// ---- DUTs/IO/PdoEntries/FSOE_340991D3.TcDUT
{attribute addProperty BoxType "EK1960-2600-0019"}
{attribute addProperty Id "FSoE_CommandUSINT811FSOUT_Module_1_Channel_1_OutputBIT10.1251FSOUT_Module_1_Channel_2_OutputBIT10.1252FSOUT_Module_1_Channel_3_OutputBIT10.1253FSOUT_Module_1_Channel_4_OutputBIT10.1254FSOUT_Module_1_ErrAckBIT10.1251FSOUT_Module_2_Channel_1_OutputBIT10.1251FSOUT_Module_2_Channel_2_OutputBIT10.1252FSOUT_Module_2_Channel_3_OutputBIT10.1253FSOUT_Module_2_Channel_4_OutputBIT10.1254FSOUT_Module_2_ErrAckBIT10.1251FSOUT_Module_3_Channel_1_OutputBIT10.1251FSOUT_Module_3_Channel_2_OutputBIT10.1252FSOUT_Module_3_Channel_3_OutputBIT10.1253FSOUT_Module_3_Channel_4_OutputBIT10.1254FSOUT_Module_3_ErrAckBIT10.1251FSOUT_Module_4_Channel_1_OutputBIT10.1251FSoE_CRC_000UINT1623FSOUT_Module_4_Channel_2_OutputBIT10.1252FSOUT_Module_4_Channel_3_OutputBIT10.1253FSOUT_Module_4_Channel_4_OutputBIT10.1254FSOUT_Module_4_ErrAckBIT10.1251FSOUT_Module_5_Channel_1_OutputBIT10.1251FSOUT_Module_5_Channel_2_OutputBIT10.1252FSOUT_Module_5_Channel_3_OutputBIT10.1253FSOUT_Module_5_Channel_4_OutputBIT10.1254FSOUT_Module_5_ErrAckBIT10.1251FSOUT_Module_6_Channel_1_OutputBIT10.1251FSOUT_Module_6_Channel_2_OutputBIT10.1252FSOUT_Module_6_Channel_3_OutputBIT10.1253FSOUT_Module_6_Channel_4_OutputBIT10.1254FSOUT_Module_6_ErrAckBIT10.1251FSOUT_Relais_Module_Channel_1_OutputBIT10.1251FSOUT_Relais_Module_Channel_2_OutputBIT10.1252FSoE_CRC_001UINT1624FSOUT_Relais_Module_Channel_3_OutputBIT10.1253FSOUT_Relais_Module_Channel_4_OutputBIT10.1254FSOUT_Relais_Module_ErrAckBIT10.1251FSIN_Module_1_ErrAckBIT10.1251FSIN_Module_2_ErrAckBIT10.1251FSIN_Module_3_ErrAckBIT10.1251FSIN_Module_4_ErrAckBIT10.1251FSIN_Module_5_ErrAckBIT10.1251FSIN_Module_6_ErrAckBIT10.1251FSIN_Module_7_ErrAckBIT10.1251FSIN_Module_8_ErrAckBIT10.1251FSIN_Module_9_ErrAck_1BIT10.1251FSIN_Module_9_ErrAck_2BIT10.1252FSIN_Module_10_ErrAck_1BIT10.1251FSIN_Module_10_ErrAck_2BIT10.1252FSoE_CRC_002UINT1625FSoE_Connection_IDUINT1622"}
{attribute addProperty CRC "873042387"}
{attribute addProperty SizeInBites "120"}
{attribute addProperty SizeInBytes "15"}
TYPE FSOE_340991D3 :
STRUCT
	{attribute addProperty Name "FSoE_Command"}
	FSoE_Command : USINT;
	{attribute addProperty Name "FSOUT_Module_1_Channel_1_Output"}
	FSOUT_Module_1_Channel_1_Output : BOOL;
	{attribute addProperty Name "FSOUT_Module_1_Channel_2_Output"}
	FSOUT_Module_1_Channel_2_Output : BOOL;
	{attribute addProperty Name "FSOUT_Module_1_Channel_3_Output"}
	FSOUT_Module_1_Channel_3_Output : BOOL;
	{attribute addProperty Name "FSOUT_Module_1_Channel_4_Output"}
	FSOUT_Module_1_Channel_4_Output : BOOL;
	{attribute addProperty Name "FSOUT_Module_1_ErrAck"}
	FSOUT_Module_1_ErrAck : BOOL;
	{attribute addProperty Name "FSOUT_Module_2_Channel_1_Output"}
	FSOUT_Module_2_Channel_1_Output : BOOL;
	{attribute addProperty Name "FSOUT_Module_2_Channel_2_Output"}
	FSOUT_Module_2_Channel_2_Output : BOOL;
	{attribute addProperty Name "FSOUT_Module_2_Channel_3_Output"}
	FSOUT_Module_2_Channel_3_Output : BOOL;
	{attribute addProperty Name "FSOUT_Module_2_Channel_4_Output"}
	FSOUT_Module_2_Channel_4_Output : BOOL;
	{attribute addProperty Name "FSOUT_Module_2_ErrAck"}
	FSOUT_Module_2_ErrAck : BOOL;
	{attribute addProperty Name "FSOUT_Module_3_Channel_1_Output"}
	FSOUT_Module_3_Channel_1_Output : BOOL;
	{attribute addProperty Name "FSOUT_Module_3_Channel_2_Output"}
	FSOUT_Module_3_Channel_2_Output : BOOL;
	{attribute addProperty Name "FSOUT_Module_3_Channel_3_Output"}
	FSOUT_Module_3_Channel_3_Output : BOOL;
	{attribute addProperty Name "FSOUT_Module_3_Channel_4_Output"}
	FSOUT_Module_3_Channel_4_Output : BOOL;
	{attribute addProperty Name "FSOUT_Module_3_ErrAck"}
	FSOUT_Module_3_ErrAck : BOOL;
	{attribute addProperty Name "FSOUT_Module_4_Channel_1_Output"}
	FSOUT_Module_4_Channel_1_Output : BOOL;
	{attribute addProperty Name "FSoE_CRC_000"}
	FSoE_CRC_000 : UINT;
	{attribute addProperty Name "FSOUT_Module_4_Channel_2_Output"}
	FSOUT_Module_4_Channel_2_Output : BOOL;
	{attribute addProperty Name "FSOUT_Module_4_Channel_3_Output"}
	FSOUT_Module_4_Channel_3_Output : BOOL;
	{attribute addProperty Name "FSOUT_Module_4_Channel_4_Output"}
	FSOUT_Module_4_Channel_4_Output : BOOL;
	{attribute addProperty Name "FSOUT_Module_4_ErrAck"}
	FSOUT_Module_4_ErrAck : BOOL;
	{attribute addProperty Name "FSOUT_Module_5_Channel_1_Output"}
	FSOUT_Module_5_Channel_1_Output : BOOL;
	{attribute addProperty Name "FSOUT_Module_5_Channel_2_Output"}
	FSOUT_Module_5_Channel_2_Output : BOOL;
	{attribute addProperty Name "FSOUT_Module_5_Channel_3_Output"}
	FSOUT_Module_5_Channel_3_Output : BOOL;
	{attribute addProperty Name "FSOUT_Module_5_Channel_4_Output"}
	FSOUT_Module_5_Channel_4_Output : BOOL;
	{attribute addProperty Name "FSOUT_Module_5_ErrAck"}
	FSOUT_Module_5_ErrAck : BOOL;
	{attribute addProperty Name "FSOUT_Module_6_Channel_1_Output"}
	FSOUT_Module_6_Channel_1_Output : BOOL;
	{attribute addProperty Name "FSOUT_Module_6_Channel_2_Output"}
	FSOUT_Module_6_Channel_2_Output : BOOL;
	{attribute addProperty Name "FSOUT_Module_6_Channel_3_Output"}
	FSOUT_Module_6_Channel_3_Output : BOOL;
	{attribute addProperty Name "FSOUT_Module_6_Channel_4_Output"}
	FSOUT_Module_6_Channel_4_Output : BOOL;
	{attribute addProperty Name "FSOUT_Module_6_ErrAck"}
	FSOUT_Module_6_ErrAck : BOOL;
	{attribute addProperty Name "FSOUT_Relais_Module_Channel_1_Output"}
	FSOUT_Relais_Module_Channel_1_Output : BOOL;
	{attribute addProperty Name "FSOUT_Relais_Module_Channel_2_Output"}
	FSOUT_Relais_Module_Channel_2_Output : BOOL;
	{attribute addProperty Name "FSoE_CRC_001"}
	FSoE_CRC_001 : UINT;
	{attribute addProperty Name "FSOUT_Relais_Module_Channel_3_Output"}
	FSOUT_Relais_Module_Channel_3_Output : BOOL;
	{attribute addProperty Name "FSOUT_Relais_Module_Channel_4_Output"}
	FSOUT_Relais_Module_Channel_4_Output : BOOL;
	{attribute addProperty Name "FSOUT_Relais_Module_ErrAck"}
	FSOUT_Relais_Module_ErrAck : BOOL;
	{attribute addProperty Name "FSIN_Module_1_ErrAck"}
	FSIN_Module_1_ErrAck : BOOL;
	{attribute addProperty Name "FSIN_Module_2_ErrAck"}
	FSIN_Module_2_ErrAck : BOOL;
	{attribute addProperty Name "FSIN_Module_3_ErrAck"}
	FSIN_Module_3_ErrAck : BOOL;
	{attribute addProperty Name "FSIN_Module_4_ErrAck"}
	FSIN_Module_4_ErrAck : BOOL;
	{attribute addProperty Name "FSIN_Module_5_ErrAck"}
	FSIN_Module_5_ErrAck : BOOL;
	{attribute addProperty Name "FSIN_Module_6_ErrAck"}
	FSIN_Module_6_ErrAck : BOOL;
	{attribute addProperty Name "FSIN_Module_7_ErrAck"}
	FSIN_Module_7_ErrAck : BOOL;
	{attribute addProperty Name "FSIN_Module_8_ErrAck"}
	FSIN_Module_8_ErrAck : BOOL;
	{attribute addProperty Name "FSIN_Module_9_ErrAck_1"}
	FSIN_Module_9_ErrAck_1 : BOOL;
	{attribute addProperty Name "FSIN_Module_9_ErrAck_2"}
	FSIN_Module_9_ErrAck_2 : BOOL;
	{attribute addProperty Name "FSIN_Module_10_ErrAck_1"}
	FSIN_Module_10_ErrAck_1 : BOOL;
	{attribute addProperty Name "FSIN_Module_10_ErrAck_2"}
	FSIN_Module_10_ErrAck_2 : BOOL;
	{attribute 'hide'}
	reserve_1 : BOOL;
	{attribute addProperty Name "FSoE_CRC_002"}
	FSoE_CRC_002 : UINT;
	{attribute addProperty Name "FSoE_Connection_ID"}
	FSoE_Connection_ID : UINT;
END_STRUCT
END_TYPE

// ---- DUTs/IO/PdoEntries/FSOE_3B47B0C1.TcDUT
{attribute addProperty BoxType "EK1960-2600-0021"}
{attribute addProperty Id "FSoE_CommandUSINT811FSOUT_Module_1_Module_FaultBIT10.1251FSOUT_Module_2_Module_FaultBIT10.1251FSOUT_Module_3_Module_FaultBIT10.1251FSOUT_Module_4_Module_FaultBIT10.1251FSOUT_Module_5_Module_FaultBIT10.1251FSOUT_Module_6_Module_FaultBIT10.1251FSOUT_Relais_Module_Module_FaultBIT10.1251FSIN_Module_1_Channel_1_Input_X6_1BIT10.1251FSIN_Module_1_Channel_2_Input_X6_2BIT10.1252FSIN_Module_1_Module_FaultBIT10.1251FSIN_Module_2_Channel_1_Input_X6_3BIT10.1251FSIN_Module_2_Channel_2_Input_X6_4BIT10.1252FSIN_Module_2_Module_FaultBIT10.1251FSIN_Module_3_Channel_1_Input_X6_5BIT10.1251FSIN_Module_3_Channel_2_Input_X6_6BIT10.1252FSIN_Module_3_Module_FaultBIT10.1251FSoE_CRC_000UINT1623FSIN_Module_4_Channel_1_Input_X6_7BIT10.1251FSIN_Module_4_Channel_2_Input_X6_8BIT10.1252FSIN_Module_4_Module_FaultBIT10.1251FSIN_Module_5_Channel_1_Input_X6_9BIT10.1251FSIN_Module_5_Channel_2_Input_X6_10BIT10.1252FSIN_Module_5_Module_FaultBIT10.1251FSIN_Module_6_Channel_1_Input_X8_1BIT10.1251FSIN_Module_6_Channel_2_Input_X8_2BIT10.1252FSIN_Module_6_Module_FaultBIT10.1251FSIN_Module_7_Channel_1_Input_X8_3BIT10.1251FSIN_Module_7_Channel_2_Input_X8_4BIT10.1252FSIN_Module_7_Module_FaultBIT10.1251FSIN_Module_8_Channel_1_Input_X8_5BIT10.1251FSIN_Module_8_Channel_2_Input_X8_6BIT10.1252FSIN_Module_8_Module_FaultBIT10.1251FSIN_Module_9_Channel_1_Input_X8_7BIT10.1251FSoE_CRC_001UINT1624FSIN_Module_9_Channel_2_Input_X8_8BIT10.1252FSIN_Module_9_Module_Fault_1BIT10.1251FSIN_Module_9_Module_Fault_2BIT10.1252FSIN_Module_10_Channel_1_Input_X8_9BIT10.1251FSIN_Module_10_Channel_2_Input_X8_10BIT10.1252FSIN_Module_10_Module_Fault_1BIT10.1251FSIN_Module_10_Module_Fault_2BIT10.1252FSoE_CRC_002UINT1625FSoE_Connection_IDUINT1622"}
{attribute addProperty CRC "994554049"}
{attribute addProperty SizeInBites "120"}
{attribute addProperty SizeInBytes "15"}
TYPE FSOE_3B47B0C1 :
STRUCT
	{attribute addProperty Name "FSoE_Command"}
	FSoE_Command : USINT;
	{attribute addProperty Name "FSOUT_Module_1_Module_Fault"}
	FSOUT_Module_1_Module_Fault : BOOL;
	{attribute addProperty Name "FSOUT_Module_2_Module_Fault"}
	FSOUT_Module_2_Module_Fault : BOOL;
	{attribute addProperty Name "FSOUT_Module_3_Module_Fault"}
	FSOUT_Module_3_Module_Fault : BOOL;
	{attribute addProperty Name "FSOUT_Module_4_Module_Fault"}
	FSOUT_Module_4_Module_Fault : BOOL;
	{attribute addProperty Name "FSOUT_Module_5_Module_Fault"}
	FSOUT_Module_5_Module_Fault : BOOL;
	{attribute addProperty Name "FSOUT_Module_6_Module_Fault"}
	FSOUT_Module_6_Module_Fault : BOOL;
	{attribute addProperty Name "FSOUT_Relais_Module_Module_Fault"}
	FSOUT_Relais_Module_Module_Fault : BOOL;
	{attribute addProperty Name "FSIN_Module_1_Channel_1_Input_X6_1"}
	FSIN_Module_1_Channel_1_Input_X6_1 : BOOL;
	{attribute addProperty Name "FSIN_Module_1_Channel_2_Input_X6_2"}
	FSIN_Module_1_Channel_2_Input_X6_2 : BOOL;
	{attribute addProperty Name "FSIN_Module_1_Module_Fault"}
	FSIN_Module_1_Module_Fault : BOOL;
	{attribute addProperty Name "FSIN_Module_2_Channel_1_Input_X6_3"}
	FSIN_Module_2_Channel_1_Input_X6_3 : BOOL;
	{attribute addProperty Name "FSIN_Module_2_Channel_2_Input_X6_4"}
	FSIN_Module_2_Channel_2_Input_X6_4 : BOOL;
	{attribute addProperty Name "FSIN_Module_2_Module_Fault"}
	FSIN_Module_2_Module_Fault : BOOL;
	{attribute addProperty Name "FSIN_Module_3_Channel_1_Input_X6_5"}
	FSIN_Module_3_Channel_1_Input_X6_5 : BOOL;
	{attribute addProperty Name "FSIN_Module_3_Channel_2_Input_X6_6"}
	FSIN_Module_3_Channel_2_Input_X6_6 : BOOL;
	{attribute addProperty Name "FSIN_Module_3_Module_Fault"}
	FSIN_Module_3_Module_Fault : BOOL;
	{attribute addProperty Name "FSoE_CRC_000"}
	FSoE_CRC_000 : UINT;
	{attribute addProperty Name "FSIN_Module_4_Channel_1_Input_X6_7"}
	FSIN_Module_4_Channel_1_Input_X6_7 : BOOL;
	{attribute addProperty Name "FSIN_Module_4_Channel_2_Input_X6_8"}
	FSIN_Module_4_Channel_2_Input_X6_8 : BOOL;
	{attribute addProperty Name "FSIN_Module_4_Module_Fault"}
	FSIN_Module_4_Module_Fault : BOOL;
	{attribute addProperty Name "FSIN_Module_5_Channel_1_Input_X6_9"}
	FSIN_Module_5_Channel_1_Input_X6_9 : BOOL;
	{attribute addProperty Name "FSIN_Module_5_Channel_2_Input_X6_10"}
	FSIN_Module_5_Channel_2_Input_X6_10 : BOOL;
	{attribute addProperty Name "FSIN_Module_5_Module_Fault"}
	FSIN_Module_5_Module_Fault : BOOL;
	{attribute addProperty Name "FSIN_Module_6_Channel_1_Input_X8_1"}
	FSIN_Module_6_Channel_1_Input_X8_1 : BOOL;
	{attribute addProperty Name "FSIN_Module_6_Channel_2_Input_X8_2"}
	FSIN_Module_6_Channel_2_Input_X8_2 : BOOL;
	{attribute addProperty Name "FSIN_Module_6_Module_Fault"}
	FSIN_Module_6_Module_Fault : BOOL;
	{attribute addProperty Name "FSIN_Module_7_Channel_1_Input_X8_3"}
	FSIN_Module_7_Channel_1_Input_X8_3 : BOOL;
	{attribute addProperty Name "FSIN_Module_7_Channel_2_Input_X8_4"}
	FSIN_Module_7_Channel_2_Input_X8_4 : BOOL;
	{attribute addProperty Name "FSIN_Module_7_Module_Fault"}
	FSIN_Module_7_Module_Fault : BOOL;
	{attribute addProperty Name "FSIN_Module_8_Channel_1_Input_X8_5"}
	FSIN_Module_8_Channel_1_Input_X8_5 : BOOL;
	{attribute addProperty Name "FSIN_Module_8_Channel_2_Input_X8_6"}
	FSIN_Module_8_Channel_2_Input_X8_6 : BOOL;
	{attribute addProperty Name "FSIN_Module_8_Module_Fault"}
	FSIN_Module_8_Module_Fault : BOOL;
	{attribute addProperty Name "FSIN_Module_9_Channel_1_Input_X8_7"}
	FSIN_Module_9_Channel_1_Input_X8_7 : BOOL;
	{attribute addProperty Name "FSoE_CRC_001"}
	FSoE_CRC_001 : UINT;
	{attribute addProperty Name "FSIN_Module_9_Channel_2_Input_X8_8"}
	FSIN_Module_9_Channel_2_Input_X8_8 : BOOL;
	{attribute addProperty Name "FSIN_Module_9_Module_Fault_1"}
	FSIN_Module_9_Module_Fault_1 : BOOL;
	{attribute addProperty Name "FSIN_Module_9_Module_Fault_2"}
	FSIN_Module_9_Module_Fault_2 : BOOL;
	{attribute addProperty Name "FSIN_Module_10_Channel_1_Input_X8_9"}
	FSIN_Module_10_Channel_1_Input_X8_9 : BOOL;
	{attribute addProperty Name "FSIN_Module_10_Channel_2_Input_X8_10"}
	FSIN_Module_10_Channel_2_Input_X8_10 : BOOL;
	{attribute addProperty Name "FSIN_Module_10_Module_Fault_1"}
	FSIN_Module_10_Module_Fault_1 : BOOL;
	{attribute addProperty Name "FSIN_Module_10_Module_Fault_2"}
	FSIN_Module_10_Module_Fault_2 : BOOL;
	{attribute 'hide'}
	reserve_1_BIT_0 : BOOL;
	{attribute 'hide'}
	reserve_1_BIT_1 : BOOL;
	{attribute 'hide'}
	reserve_1_BIT_2 : BOOL;
	{attribute 'hide'}
	reserve_1_BIT_3 : BOOL;
	{attribute 'hide'}
	reserve_1_BIT_4 : BOOL;
	{attribute 'hide'}
	reserve_1_BIT_5 : BOOL;
	{attribute 'hide'}
	reserve_1_BIT_6 : BOOL;
	{attribute 'hide'}
	reserve_1_BIT_7 : BOOL;
	{attribute 'hide'}
	reserve_1_BIT_8 : BOOL;
	{attribute addProperty Name "FSoE_CRC_002"}
	FSoE_CRC_002 : UINT;
	{attribute addProperty Name "FSoE_Connection_ID"}
	FSoE_Connection_ID : UINT;
END_STRUCT
END_TYPE

// ---- DUTs/IO/PdoEntries/FSOE_9F057372.TcDUT
{attribute addProperty BoxType "EK1960-2600-0021"}
{attribute addProperty Id "FSoE_CommandUSINT811FSOUT_Module_1_Channel_1_Output_X5_1BIT10.1251FSOUT_Module_1_Channel_2_Output_X5_2BIT10.1252FSOUT_Module_1_Channel_3_Output_X5_3BIT10.1253FSOUT_Module_1_Channel_4_Output_X5_4BIT10.1254FSOUT_Module_1_ErrAckBIT10.1251FSOUT_Module_2_Channel_1_Output_X5_5BIT10.1251FSOUT_Module_2_Channel_2_Output_X5_6BIT10.1252FSOUT_Module_2_Channel_3_Output_X5_7BIT10.1253FSOUT_Module_2_Channel_4_Output_X5_8BIT10.1254FSOUT_Module_2_ErrAckBIT10.1251FSOUT_Module_3_Channel_1_Output_X7_1BIT10.1251FSOUT_Module_3_Channel_2_Output_X7_2BIT10.1252FSOUT_Module_3_Channel_3_Output_X7_3BIT10.1253FSOUT_Module_3_Channel_4_Output_X7_4BIT10.1254FSOUT_Module_3_ErrAckBIT10.1251FSOUT_Module_4_Channel_1_Output_X7_5BIT10.1251FSoE_CRC_000UINT1623FSOUT_Module_4_Channel_2_Output_X7_6BIT10.1252FSOUT_Module_4_Channel_3_Output_X7_7BIT10.1253FSOUT_Module_4_Channel_4_Output_X7_8BIT10.1254FSOUT_Module_4_ErrAckBIT10.1251FSOUT_Module_5_Channel_1_Output_X9_1BIT10.1251FSOUT_Module_5_Channel_2_Output_X9_2BIT10.1252FSOUT_Module_5_Channel_3_Output_X9_3BIT10.1253FSOUT_Module_5_Channel_4_Output_X9_4BIT10.1254FSOUT_Module_5_ErrAckBIT10.1251FSOUT_Module_6_Channel_1_Output_X9_5BIT10.1251FSOUT_Module_6_Channel_2_Output_X9_6BIT10.1252FSOUT_Module_6_Channel_3_Output_X9_7BIT10.1253FSOUT_Module_6_Channel_4_Output_X9_8BIT10.1254FSOUT_Module_6_ErrAckBIT10.1251FSOUT_Relais_Module_Channel_1_Output_X4_1_X4_5BIT10.1251FSOUT_Relais_Module_Channel_2_Output_X4_2_X4_6BIT10.1252FSoE_CRC_001UINT1624FSOUT_Relais_Module_Channel_3_Output_X4_3_X4_7BIT10.1253FSOUT_Relais_Module_Channel_4_Output_X4_4_X4_8BIT10.1254FSOUT_Relais_Module_ErrAckBIT10.1251FSIN_Module_1_ErrAckBIT10.1251FSIN_Module_2_ErrAckBIT10.1251FSIN_Module_3_ErrAckBIT10.1251FSIN_Module_4_ErrAckBIT10.1251FSIN_Module_5_ErrAckBIT10.1251FSIN_Module_6_ErrAckBIT10.1251FSIN_Module_7_ErrAckBIT10.1251FSIN_Module_8_ErrAckBIT10.1251FSIN_Module_9_Err_Ack_1BIT10.1251FSIN_Module_9_Err_Ack_2BIT10.1252FSIN_Module_10_Err_Ack_1BIT10.1251FSIN_Module_10_Err_Ack_2BIT10.1252FSoE_CRC_002UINT1625FSoE_Connection_IDUINT1622"}
{attribute addProperty CRC "2667934578"}
{attribute addProperty SizeInBites "120"}
{attribute addProperty SizeInBytes "15"}
TYPE FSOE_9F057372 :
STRUCT
	{attribute addProperty Name "FSoE_Command"}
	FSoE_Command : USINT;
	{attribute addProperty Name "FSOUT_Module_1_Channel_1_Output_X5_1"}
	FSOUT_Module_1_Channel_1_Output_X5_1 : BOOL;
	{attribute addProperty Name "FSOUT_Module_1_Channel_2_Output_X5_2"}
	FSOUT_Module_1_Channel_2_Output_X5_2 : BOOL;
	{attribute addProperty Name "FSOUT_Module_1_Channel_3_Output_X5_3"}
	FSOUT_Module_1_Channel_3_Output_X5_3 : BOOL;
	{attribute addProperty Name "FSOUT_Module_1_Channel_4_Output_X5_4"}
	FSOUT_Module_1_Channel_4_Output_X5_4 : BOOL;
	{attribute addProperty Name "FSOUT_Module_1_ErrAck"}
	FSOUT_Module_1_ErrAck : BOOL;
	{attribute addProperty Name "FSOUT_Module_2_Channel_1_Output_X5_5"}
	FSOUT_Module_2_Channel_1_Output_X5_5 : BOOL;
	{attribute addProperty Name "FSOUT_Module_2_Channel_2_Output_X5_6"}
	FSOUT_Module_2_Channel_2_Output_X5_6 : BOOL;
	{attribute addProperty Name "FSOUT_Module_2_Channel_3_Output_X5_7"}
	FSOUT_Module_2_Channel_3_Output_X5_7 : BOOL;
	{attribute addProperty Name "FSOUT_Module_2_Channel_4_Output_X5_8"}
	FSOUT_Module_2_Channel_4_Output_X5_8 : BOOL;
	{attribute addProperty Name "FSOUT_Module_2_ErrAck"}
	FSOUT_Module_2_ErrAck : BOOL;
	{attribute addProperty Name "FSOUT_Module_3_Channel_1_Output_X7_1"}
	FSOUT_Module_3_Channel_1_Output_X7_1 : BOOL;
	{attribute addProperty Name "FSOUT_Module_3_Channel_2_Output_X7_2"}
	FSOUT_Module_3_Channel_2_Output_X7_2 : BOOL;
	{attribute addProperty Name "FSOUT_Module_3_Channel_3_Output_X7_3"}
	FSOUT_Module_3_Channel_3_Output_X7_3 : BOOL;
	{attribute addProperty Name "FSOUT_Module_3_Channel_4_Output_X7_4"}
	FSOUT_Module_3_Channel_4_Output_X7_4 : BOOL;
	{attribute addProperty Name "FSOUT_Module_3_ErrAck"}
	FSOUT_Module_3_ErrAck : BOOL;
	{attribute addProperty Name "FSOUT_Module_4_Channel_1_Output_X7_5"}
	FSOUT_Module_4_Channel_1_Output_X7_5 : BOOL;
	{attribute addProperty Name "FSoE_CRC_000"}
	FSoE_CRC_000 : UINT;
	{attribute addProperty Name "FSOUT_Module_4_Channel_2_Output_X7_6"}
	FSOUT_Module_4_Channel_2_Output_X7_6 : BOOL;
	{attribute addProperty Name "FSOUT_Module_4_Channel_3_Output_X7_7"}
	FSOUT_Module_4_Channel_3_Output_X7_7 : BOOL;
	{attribute addProperty Name "FSOUT_Module_4_Channel_4_Output_X7_8"}
	FSOUT_Module_4_Channel_4_Output_X7_8 : BOOL;
	{attribute addProperty Name "FSOUT_Module_4_ErrAck"}
	FSOUT_Module_4_ErrAck : BOOL;
	{attribute addProperty Name "FSOUT_Module_5_Channel_1_Output_X9_1"}
	FSOUT_Module_5_Channel_1_Output_X9_1 : BOOL;
	{attribute addProperty Name "FSOUT_Module_5_Channel_2_Output_X9_2"}
	FSOUT_Module_5_Channel_2_Output_X9_2 : BOOL;
	{attribute addProperty Name "FSOUT_Module_5_Channel_3_Output_X9_3"}
	FSOUT_Module_5_Channel_3_Output_X9_3 : BOOL;
	{attribute addProperty Name "FSOUT_Module_5_Channel_4_Output_X9_4"}
	FSOUT_Module_5_Channel_4_Output_X9_4 : BOOL;
	{attribute addProperty Name "FSOUT_Module_5_ErrAck"}
	FSOUT_Module_5_ErrAck : BOOL;
	{attribute addProperty Name "FSOUT_Module_6_Channel_1_Output_X9_5"}
	FSOUT_Module_6_Channel_1_Output_X9_5 : BOOL;
	{attribute addProperty Name "FSOUT_Module_6_Channel_2_Output_X9_6"}
	FSOUT_Module_6_Channel_2_Output_X9_6 : BOOL;
	{attribute addProperty Name "FSOUT_Module_6_Channel_3_Output_X9_7"}
	FSOUT_Module_6_Channel_3_Output_X9_7 : BOOL;
	{attribute addProperty Name "FSOUT_Module_6_Channel_4_Output_X9_8"}
	FSOUT_Module_6_Channel_4_Output_X9_8 : BOOL;
	{attribute addProperty Name "FSOUT_Module_6_ErrAck"}
	FSOUT_Module_6_ErrAck : BOOL;
	{attribute addProperty Name "FSOUT_Relais_Module_Channel_1_Output_X4_1_X4_5"}
	FSOUT_Relais_Module_Channel_1_Output_X4_1_X4_5 : BOOL;
	{attribute addProperty Name "FSOUT_Relais_Module_Channel_2_Output_X4_2_X4_6"}
	FSOUT_Relais_Module_Channel_2_Output_X4_2_X4_6 : BOOL;
	{attribute addProperty Name "FSoE_CRC_001"}
	FSoE_CRC_001 : UINT;
	{attribute addProperty Name "FSOUT_Relais_Module_Channel_3_Output_X4_3_X4_7"}
	FSOUT_Relais_Module_Channel_3_Output_X4_3_X4_7 : BOOL;
	{attribute addProperty Name "FSOUT_Relais_Module_Channel_4_Output_X4_4_X4_8"}
	FSOUT_Relais_Module_Channel_4_Output_X4_4_X4_8 : BOOL;
	{attribute addProperty Name "FSOUT_Relais_Module_ErrAck"}
	FSOUT_Relais_Module_ErrAck : BOOL;
	{attribute addProperty Name "FSIN_Module_1_ErrAck"}
	FSIN_Module_1_ErrAck : BOOL;
	{attribute addProperty Name "FSIN_Module_2_ErrAck"}
	FSIN_Module_2_ErrAck : BOOL;
	{attribute addProperty Name "FSIN_Module_3_ErrAck"}
	FSIN_Module_3_ErrAck : BOOL;
	{attribute addProperty Name "FSIN_Module_4_ErrAck"}
	FSIN_Module_4_ErrAck : BOOL;
	{attribute addProperty Name "FSIN_Module_5_ErrAck"}
	FSIN_Module_5_ErrAck : BOOL;
	{attribute addProperty Name "FSIN_Module_6_ErrAck"}
	FSIN_Module_6_ErrAck : BOOL;
	{attribute addProperty Name "FSIN_Module_7_ErrAck"}
	FSIN_Module_7_ErrAck : BOOL;
	{attribute addProperty Name "FSIN_Module_8_ErrAck"}
	FSIN_Module_8_ErrAck : BOOL;
	{attribute addProperty Name "FSIN_Module_9_Err_Ack_1"}
	FSIN_Module_9_Err_Ack_1 : BOOL;
	{attribute addProperty Name "FSIN_Module_9_Err_Ack_2"}
	FSIN_Module_9_Err_Ack_2 : BOOL;
	{attribute addProperty Name "FSIN_Module_10_Err_Ack_1"}
	FSIN_Module_10_Err_Ack_1 : BOOL;
	{attribute addProperty Name "FSIN_Module_10_Err_Ack_2"}
	FSIN_Module_10_Err_Ack_2 : BOOL;
	{attribute 'hide'}
	reserve_1 : BOOL;
	{attribute addProperty Name "FSoE_CRC_002"}
	FSoE_CRC_002 : UINT;
	{attribute addProperty Name "FSoE_Connection_ID"}
	FSoE_Connection_ID : UINT;
END_STRUCT
END_TYPE

// ---- DUTs/IO/PDOs/InfoData_192954DE.TcDUT
{attribute addProperty BoxType "EK1100-0000-0018"}
{attribute addProperty Id "StateAT %I*UINT1620"}
{attribute addProperty CRC "422139102"}
{attribute addProperty SizeInBites "16"}
{attribute addProperty SizeInBytes "2"}
TYPE InfoData_192954DE :
STRUCT
	{attribute addProperty Name "State"}
	State AT %I* : UINT;
END_STRUCT
END_TYPE

// ---- DUTs/IO/PDOs/WcState_28A86775.TcDUT
{attribute addProperty BoxType "EJ1101-0022-0016"}
{attribute addProperty Id "WcStateAT %I*BIT10.1250"}
{attribute addProperty CRC "682125173"}
{attribute addProperty SizeInBites "1"}
{attribute addProperty SizeInBytes "0.125"}
TYPE WcState_28A86775 :
STRUCT
	{attribute addProperty Name "WcState"}
	WcState AT %I* : BOOL;
END_STRUCT
END_TYPE

// ---- DUTs/IO/PDOs/InfoData_BC63D37F.TcDUT
{attribute addProperty BoxType "EJ1101-0022-0016"}
{attribute addProperty Id "AdsAddrAT %I*AMSADDR6480StateAT %I*UINT1620"}
{attribute addProperty CRC "3160658815"}
{attribute addProperty SizeInBites "80"}
{attribute addProperty SizeInBytes "10"}
TYPE InfoData_BC63D37F :
STRUCT
	{attribute addProperty Name "AdsAddr"}
	AdsAddr AT %I* : AMSADDR;
	{attribute addProperty Name "State"}
	State AT %I* : UINT;
END_STRUCT
END_TYPE

// ---- DUTs/IO/PDOs/Channel_E4AEF59E.TcDUT
{attribute addProperty BoxType "EJ1008-0000-0017"}
{attribute addProperty Id "InputAT %I*BOOL81"}
{attribute addProperty CRC "3836671390"}
{attribute addProperty SizeInBites "8"}
{attribute addProperty SizeInBytes "1"}
TYPE Channel_E4AEF59E :
STRUCT
	{attribute addProperty Name "Input"}
	Input AT %I* : BOOL;
END_STRUCT
END_TYPE

// ---- DUTs/IO/PDOs/WcState_98A4DF75.TcDUT
{attribute addProperty BoxType "EJ1008-0000-0017"}
{attribute addProperty Id "WcStateAT %I*BIT10.1250InputToggleAT %I*BIT10.1250"}
{attribute addProperty CRC "2560941941"}
{attribute addProperty SizeInBites "2"}
{attribute addProperty SizeInBytes "0.25"}
TYPE WcState_98A4DF75 :
STRUCT
	{attribute addProperty Name "WcState"}
	WcState AT %I* : BOOL;
	{attribute addProperty Name "InputToggle"}
	InputToggle AT %I* : BOOL;
END_STRUCT
END_TYPE

// ---- DUTs/IO/PDOs/Channel_7F374EB0.TcDUT
{attribute addProperty BoxType "EJ1859-0000-0017"}
{attribute addProperty Id "OutputAT %Q*BOOL81"}
{attribute addProperty CRC "2134331056"}
{attribute addProperty SizeInBites "8"}
{attribute addProperty SizeInBytes "1"}
TYPE Channel_7F374EB0 :
STRUCT
	{attribute addProperty Name "Output"}
	Output AT %Q* : BOOL;
END_STRUCT
END_TYPE

// ---- DUTs/IO/PDOs/PWM_Outputs_Channel_A83D42AA.TcDUT
{attribute addProperty BoxType "EJ2502-0000-0023"}
{attribute addProperty Id "PWM_outputAT %Q*UINT162"}
{attribute addProperty CRC "2822587050"}
{attribute addProperty SizeInBites "16"}
{attribute addProperty SizeInBytes "2"}
TYPE PWM_Outputs_Channel_A83D42AA :
STRUCT
	{attribute addProperty Name "PWM_output"}
	PWM_output AT %Q* : UINT;
END_STRUCT
END_TYPE

// ---- DUTs/IO/PDOs/PTO_Status_B9BB57FE.TcDUT
{attribute addProperty BoxType "EJ2521-0224-0016"}
{attribute addProperty Id "StatusAT %I*Status_30784993162"}
{attribute addProperty CRC "3116062718"}
{attribute addProperty SizeInBites "16"}
{attribute addProperty SizeInBytes "2"}
TYPE PTO_Status_B9BB57FE :
STRUCT
	{attribute addProperty Name "Status"}
	Status AT %I* : Status_30784993;
END_STRUCT
END_TYPE

// ---- DUTs/IO/PDOs/ENC_Status_compact_FA080ECA.TcDUT
{attribute addProperty BoxType "EJ2521-0224-0016"}
{attribute addProperty Id "StatusAT %I*Status_F22324A31620Counter_valueAT %I*UINT16217Latch_valueAT %I*UINT16218"}
{attribute addProperty CRC "4194832074"}
{attribute addProperty SizeInBites "48"}
{attribute addProperty SizeInBytes "6"}
TYPE ENC_Status_compact_FA080ECA :
STRUCT
	{attribute addProperty Name "Status"}
	Status AT %I* : Status_F22324A3;
	{attribute addProperty Name "Counter_value"}
	Counter_value AT %I* : UINT;
	{attribute addProperty Name "Latch_value"}
	Latch_value AT %I* : UINT;
END_STRUCT
END_TYPE

// ---- DUTs/IO/PDOs/PLS_Status_Channel_7A2392D1.TcDUT
{attribute addProperty BoxType "EJ2521-0224-0016"}
{attribute addProperty Id "StatusAT %I*Status_2B4F1F8E162"}
{attribute addProperty CRC "2049151697"}
{attribute addProperty SizeInBites "16"}
{attribute addProperty SizeInBytes "2"}
TYPE PLS_Status_Channel_7A2392D1 :
STRUCT
	{attribute addProperty Name "Status"}
	Status AT %I* : Status_2B4F1F8E;
END_STRUCT
END_TYPE

// ---- DUTs/IO/PDOs/PTO_Control_0A6210C3.TcDUT
{attribute addProperty BoxType "EJ2521-0224-0016"}
{attribute addProperty Id "ControlAT %Q*Control_A1EB0E501621Frequency_valueAT %Q*UINT16217"}
{attribute addProperty CRC "174198979"}
{attribute addProperty SizeInBites "32"}
{attribute addProperty SizeInBytes "4"}
TYPE PTO_Control_0A6210C3 :
STRUCT
	{attribute addProperty Name "Control"}
	Control AT %Q* : Control_A1EB0E50;
	{attribute addProperty Name "Frequency_value"}
	Frequency_value AT %Q* : UINT;
END_STRUCT
END_TYPE

// ---- DUTs/IO/PDOs/PTO_Target_compact_C80C22BB.TcDUT
{attribute addProperty BoxType "EJ2521-0224-0016"}
{attribute addProperty Id "Target_counter_valueAT %Q*UINT162"}
{attribute addProperty CRC "3356238523"}
{attribute addProperty SizeInBites "16"}
{attribute addProperty SizeInBytes "2"}
TYPE PTO_Target_compact_C80C22BB :
STRUCT
	{attribute addProperty Name "Target_counter_value"}
	Target_counter_value AT %Q* : UINT;
END_STRUCT
END_TYPE

// ---- DUTs/IO/PDOs/ENC_Control_compact_5C86AA9D.TcDUT
{attribute addProperty BoxType "EJ2521-0224-0016"}
{attribute addProperty Id "ControlAT %Q*Control_E8AFF3DF1620Set_counter_valueAT %Q*UINT16217"}
{attribute addProperty CRC "1552329373"}
{attribute addProperty SizeInBites "32"}
{attribute addProperty SizeInBytes "4"}
TYPE ENC_Control_compact_5C86AA9D :
STRUCT
	{attribute addProperty Name "Control"}
	Control AT %Q* : Control_E8AFF3DF;
	{attribute addProperty Name "Set_counter_value"}
	Set_counter_value AT %Q* : UINT;
END_STRUCT
END_TYPE

// ---- DUTs/IO/PDOs/PLS_Control_compact_Channel_F7E9C674.TcDUT
{attribute addProperty BoxType "EJ2521-0224-0016"}
{attribute addProperty Id "ControlAT %Q*Control_055E5E7E1621Switch_on_valueAT %Q*UINT16217Switch_off_valueAT %Q*UINT16218"}
{attribute addProperty CRC "4159293044"}
{attribute addProperty SizeInBites "48"}
{attribute addProperty SizeInBytes "6"}
TYPE PLS_Control_compact_Channel_F7E9C674 :
STRUCT
	{attribute addProperty Name "Control"}
	Control AT %Q* : Control_055E5E7E;
	{attribute addProperty Name "Switch_on_value"}
	Switch_on_value AT %Q* : UINT;
	{attribute addProperty Name "Switch_off_value"}
	Switch_off_value AT %Q* : UINT;
END_STRUCT
END_TYPE

// ---- DUTs/IO/PDOs/PTO_Status_Channel_B9BB57FE.TcDUT
{attribute addProperty BoxType "EJ2522-0000-0022"}
{attribute addProperty Id "StatusAT %I*Status_30784993162"}
{attribute addProperty CRC "3116062718"}
{attribute addProperty SizeInBites "16"}
{attribute addProperty SizeInBytes "2"}
TYPE PTO_Status_Channel_B9BB57FE :
STRUCT
	{attribute addProperty Name "Status"}
	Status AT %I* : Status_30784993;
END_STRUCT
END_TYPE

// ---- DUTs/IO/PDOs/ENC_Status_Channel_D7F89173.TcDUT
{attribute addProperty BoxType "EJ2522-0000-0022"}
{attribute addProperty Id "StatusAT %I*Status_2BCA7A521620Counter_valueAT %I*UDINT32417"}
{attribute addProperty CRC "3623391603"}
{attribute addProperty SizeInBites "48"}
{attribute addProperty SizeInBytes "6"}
TYPE ENC_Status_Channel_D7F89173 :
STRUCT
	{attribute addProperty Name "Status"}
	Status AT %I* : Status_2BCA7A52;
	{attribute addProperty Name "Counter_value"}
	Counter_value AT %I* : UDINT;
END_STRUCT
END_TYPE

// ---- DUTs/IO/PDOs/PTO_Control_Channel_0A6210C3.TcDUT
{attribute addProperty BoxType "EJ2522-0000-0022"}
{attribute addProperty Id "ControlAT %Q*Control_A1EB0E501621Frequency_valueAT %Q*UINT16217"}
{attribute addProperty CRC "174198979"}
{attribute addProperty SizeInBites "32"}
{attribute addProperty SizeInBytes "4"}
TYPE PTO_Control_Channel_0A6210C3 :
STRUCT
	{attribute addProperty Name "Control"}
	Control AT %Q* : Control_A1EB0E50;
	{attribute addProperty Name "Frequency_value"}
	Frequency_value AT %Q* : UINT;
END_STRUCT
END_TYPE

// ---- DUTs/IO/PDOs/PTO_Target_Channel_3945899C.TcDUT
{attribute addProperty BoxType "EJ2522-0000-0022"}
{attribute addProperty Id "Target_counter_valueAT %Q*UDINT324"}
{attribute addProperty CRC "960858524"}
{attribute addProperty SizeInBites "32"}
{attribute addProperty SizeInBytes "4"}
TYPE PTO_Target_Channel_3945899C :
STRUCT
	{attribute addProperty Name "Target_counter_value"}
	Target_counter_value AT %Q* : UDINT;
END_STRUCT
END_TYPE

// ---- DUTs/IO/PDOs/ENC_Control_Channel_8309D56E.TcDUT
{attribute addProperty BoxType "EJ2522-0000-0022"}
{attribute addProperty Id "ControlAT %Q*Control_A79237B31620Set_counter_valueAT %Q*UDINT32417"}
{attribute addProperty CRC "2198459758"}
{attribute addProperty SizeInBites "48"}
{attribute addProperty SizeInBytes "6"}
TYPE ENC_Control_Channel_8309D56E :
STRUCT
	{attribute addProperty Name "Control"}
	Control AT %Q* : Control_A79237B3;
	{attribute addProperty Name "Set_counter_value"}
	Set_counter_value AT %Q* : UDINT;
END_STRUCT
END_TYPE

// ---- DUTs/IO/PDOs/AI_Standard_Channel_5763EEB9.TcDUT
{attribute addProperty BoxType "EJ3004-0000-0019"}
{attribute addProperty Id "StatusAT %I*Status_C6F82E6F1621ValueAT %I*INT16217"}
{attribute addProperty CRC "1466166969"}
{attribute addProperty SizeInBites "32"}
{attribute addProperty SizeInBytes "4"}
TYPE AI_Standard_Channel_5763EEB9 :
STRUCT
	{attribute addProperty Name "Status"}
	Status AT %I* : Status_C6F82E6F;
	{attribute addProperty Name "Value"}
	Value AT %I* : INT;
END_STRUCT
END_TYPE

// ---- DUTs/IO/PDOs/AI_Standard_Channel_F16A160D.TcDUT
{attribute addProperty BoxType "EJ3004-0000-0020"}
{attribute addProperty Id "StatusAT %I*Status_F0C7FE3C1621ValueAT %I*INT16217"}
{attribute addProperty CRC "4050261517"}
{attribute addProperty SizeInBites "32"}
{attribute addProperty SizeInBytes "4"}
TYPE AI_Standard_Channel_F16A160D :
STRUCT
	{attribute addProperty Name "Status"}
	Status AT %I* : Status_F0C7FE3C;
	{attribute addProperty Name "Value"}
	Value AT %I* : INT;
END_STRUCT
END_TYPE

// ---- DUTs/IO/PDOs/AI_Standard_Channel_087F71C7.TcDUT
{attribute addProperty BoxType "EJ3104-0000-0019"}
{attribute addProperty Id "StatusAT %I*Status_845218981621ValueAT %I*INT16217"}
{attribute addProperty CRC "142569927"}
{attribute addProperty SizeInBites "32"}
{attribute addProperty SizeInBytes "4"}
TYPE AI_Standard_Channel_087F71C7 :
STRUCT
	{attribute addProperty Name "Status"}
	Status AT %I* : Status_84521898;
	{attribute addProperty Name "Value"}
	Value AT %I* : INT;
END_STRUCT
END_TYPE

// ---- DUTs/IO/PDOs/RTD_Inputs_Channel_5763EEB9.TcDUT
{attribute addProperty BoxType "EJ3202-0000-0019"}
{attribute addProperty Id "StatusAT %I*Status_C6F82E6F1621ValueAT %I*INT16217"}
{attribute addProperty CRC "1466166969"}
{attribute addProperty SizeInBites "32"}
{attribute addProperty SizeInBytes "4"}
TYPE RTD_Inputs_Channel_5763EEB9 :
STRUCT
	{attribute addProperty Name "Status"}
	Status AT %I* : Status_C6F82E6F;
	{attribute addProperty Name "Value"}
	Value AT %I* : INT;
END_STRUCT
END_TYPE

// ---- DUTs/IO/PDOs/RTD_Inputs_Channel_17AE08DB.TcDUT
{attribute addProperty BoxType "EJ3214-0000-0016"}
{attribute addProperty Id "StatusAT %I*Status_C3A5DD7C1621ValueAT %I*INT16217"}
{attribute addProperty CRC "397281499"}
{attribute addProperty SizeInBites "32"}
{attribute addProperty SizeInBytes "4"}
TYPE RTD_Inputs_Channel_17AE08DB :
STRUCT
	{attribute addProperty Name "Status"}
	Status AT %I* : Status_C3A5DD7C;
	{attribute addProperty Name "Value"}
	Value AT %I* : INT;
END_STRUCT
END_TYPE

// ---- DUTs/IO/PDOs/TC_Channel_17AE08DB.TcDUT
{attribute addProperty BoxType "EJ3318-0000-0017"}
{attribute addProperty Id "StatusAT %I*Status_C3A5DD7C1621ValueAT %I*INT16217"}
{attribute addProperty CRC "397281499"}
{attribute addProperty SizeInBites "32"}
{attribute addProperty SizeInBytes "4"}
TYPE TC_Channel_17AE08DB :
STRUCT
	{attribute addProperty Name "Status"}
	Status AT %I* : Status_C3A5DD7C;
	{attribute addProperty Name "Value"}
	Value AT %I* : INT;
END_STRUCT
END_TYPE

// ---- DUTs/IO/PDOs/AO_Outputs_Channel_F57FA4F9.TcDUT
{attribute addProperty BoxType "EJ4002-0000-0017"}
{attribute addProperty Id "Analog_outputAT %Q*INT162"}
{attribute addProperty CRC "4118783225"}
{attribute addProperty SizeInBites "16"}
{attribute addProperty SizeInBytes "2"}
TYPE AO_Outputs_Channel_F57FA4F9 :
STRUCT
	{attribute addProperty Name "Analog_output"}
	Analog_output AT %Q* : INT;
END_STRUCT
END_TYPE

// ---- DUTs/IO/PDOs/AO_Output_Channel_F57FA4F9.TcDUT
{attribute addProperty BoxType "EJ4002-0000-0018"}
{attribute addProperty Id "Analog_outputAT %Q*INT162"}
{attribute addProperty CRC "4118783225"}
{attribute addProperty SizeInBites "16"}
{attribute addProperty SizeInBytes "2"}
TYPE AO_Output_Channel_F57FA4F9 :
STRUCT
	{attribute addProperty Name "Analog_output"}
	Analog_output AT %Q* : INT;
END_STRUCT
END_TYPE

// ---- DUTs/IO/PDOs/SSI_Inputs_Channel_F7D238D1.TcDUT
{attribute addProperty BoxType "EJ5002-0000-0016"}
{attribute addProperty Id "StatusAT %I*Status_3D859DDA1621Counter_valueAT %I*UDINT32417"}
{attribute addProperty CRC "4157749457"}
{attribute addProperty SizeInBites "48"}
{attribute addProperty SizeInBytes "6"}
TYPE SSI_Inputs_Channel_F7D238D1 :
STRUCT
	{attribute addProperty Name "Status"}
	Status AT %I* : Status_3D859DDA;
	{attribute addProperty Name "Counter_value"}
	Counter_value AT %I* : UDINT;
END_STRUCT
END_TYPE

// ---- DUTs/IO/PDOs/SSI_Inputs_Channel_32C7114D.TcDUT
{attribute addProperty BoxType "EJ5002-0000-0017"}
{attribute addProperty Id "StatusAT %I*Status_F6CF9E121621Counter_valueAT %I*UDINT32417"}
{attribute addProperty CRC "851906893"}
{attribute addProperty SizeInBites "48"}
{attribute addProperty SizeInBytes "6"}
TYPE SSI_Inputs_Channel_32C7114D :
STRUCT
	{attribute addProperty Name "Status"}
	Status AT %I* : Status_F6CF9E12;
	{attribute addProperty Name "Counter_value"}
	Counter_value AT %I* : UDINT;
END_STRUCT
END_TYPE

// ---- DUTs/IO/PDOs/ENC_Status_compact_5BAFF8F5.TcDUT
{attribute addProperty BoxType "EJ5101-0000-0016"}
{attribute addProperty Id "StatusAT %I*Status_F0C09FF11621Counter_valueAT %I*UINT16217Latch_valueAT %I*UINT16218"}
{attribute addProperty CRC "1538259189"}
{attribute addProperty SizeInBites "48"}
{attribute addProperty SizeInBytes "6"}
TYPE ENC_Status_compact_5BAFF8F5 :
STRUCT
	{attribute addProperty Name "Status"}
	Status AT %I* : Status_F0C09FF1;
	{attribute addProperty Name "Counter_value"}
	Counter_value AT %I* : UINT;
	{attribute addProperty Name "Latch_value"}
	Latch_value AT %I* : UINT;
END_STRUCT
END_TYPE

// ---- DUTs/IO/PDOs/ENC_Control_compact_03701F33.TcDUT
{attribute addProperty BoxType "EJ5101-0000-0016"}
{attribute addProperty Id "ControlAT %Q*Control_38B054C81621Set_counter_valueAT %Q*UINT16217"}
{attribute addProperty CRC "57679667"}
{attribute addProperty SizeInBites "32"}
{attribute addProperty SizeInBytes "4"}
TYPE ENC_Control_compact_03701F33 :
STRUCT
	{attribute addProperty Name "Control"}
	Control AT %Q* : Control_38B054C8;
	{attribute addProperty Name "Set_counter_value"}
	Set_counter_value AT %Q* : UINT;
END_STRUCT
END_TYPE

// ---- DUTs/IO/PDOs/ENC_Inputs_001F11BA.TcDUT
{attribute addProperty BoxType "EJ5151-0000-0016"}
{attribute addProperty Id "StatusAT %I*Status_BAC5C70E1621Counter_valueAT %I*UINT16217Latch_valueAT %I*UINT16218"}
{attribute addProperty CRC "2036154"}
{attribute addProperty SizeInBites "48"}
{attribute addProperty SizeInBytes "6"}
TYPE ENC_Inputs_001F11BA :
STRUCT
	{attribute addProperty Name "Status"}
	Status AT %I* : Status_BAC5C70E;
	{attribute addProperty Name "Counter_value"}
	Counter_value AT %I* : UINT;
	{attribute addProperty Name "Latch_value"}
	Latch_value AT %I* : UINT;
END_STRUCT
END_TYPE

// ---- DUTs/IO/PDOs/ENC_Inputs_AC51B8A0.TcDUT
{attribute addProperty BoxType "EJ5151-0000-0016"}
{attribute addProperty Id "Period_valueAT %I*UDINT324"}
{attribute addProperty CRC "2891036832"}
{attribute addProperty SizeInBites "32"}
{attribute addProperty SizeInBytes "4"}
TYPE ENC_Inputs_AC51B8A0 :
STRUCT
	{attribute addProperty Name "Period_value"}
	Period_value AT %I* : UDINT;
END_STRUCT
END_TYPE

// ---- DUTs/IO/PDOs/ENC_Outputs_03701F33.TcDUT
{attribute addProperty BoxType "EJ5151-0000-0016"}
{attribute addProperty Id "ControlAT %Q*Control_38B054C81621Set_counter_valueAT %Q*UINT16217"}
{attribute addProperty CRC "57679667"}
{attribute addProperty SizeInBites "32"}
{attribute addProperty SizeInBytes "4"}
TYPE ENC_Outputs_03701F33 :
STRUCT
	{attribute addProperty Name "Control"}
	Control AT %Q* : Control_38B054C8;
	{attribute addProperty Name "Set_counter_value"}
	Set_counter_value AT %Q* : UINT;
END_STRUCT
END_TYPE

// ---- DUTs/IO/PDOs/COM_Inputs_Channel_85D1D733.TcDUT
{attribute addProperty BoxType "EJ6002-0000-0016"}
{attribute addProperty Id "StatusAT %I*Status_0CBEDEF81621Data_InAT %I*ARRAY[0 ..21] OF USINT176220"}
{attribute addProperty CRC "3699519399"}
{attribute addProperty SizeInBites "192"}
{attribute addProperty SizeInBytes "24"}
TYPE COM_Inputs_Channel_85D1D733 :
STRUCT
	{attribute addProperty Name "Status"}
	Status AT %I* : Status_0CBEDEF8;
	{attribute addProperty Name "Data_In"}
	Data_In AT %I* : ARRAY[0 ..21] OF USINT;
END_STRUCT
END_TYPE

// ---- DUTs/IO/PDOs/COM_Outputs_Channel_85BCA431.TcDUT
{attribute addProperty BoxType "EJ6002-0000-0016"}
{attribute addProperty Id "CtrlAT %Q*Ctrl_9717E3671621Data_OutAT %Q*ARRAY[0 ..21] OF USINT176220"}
{attribute addProperty CRC "604386845"}
{attribute addProperty SizeInBites "192"}
{attribute addProperty SizeInBytes "24"}
TYPE COM_Outputs_Channel_85BCA431 :
STRUCT
	{attribute addProperty Name "Ctrl"}
	Ctrl AT %Q* : Ctrl_9717E367;
	{attribute addProperty Name "Data_Out"}
	Data_Out AT %Q* : ARRAY[0 ..21] OF USINT;
END_STRUCT
END_TYPE

// ---- DUTs/IO/PDOs/DeviceState_Inputs_Device_345DC0EE.TcDUT
{attribute addProperty BoxType "EJ6224-0000-0016"}
{attribute addProperty Id "Device_DiagAT %I*BOOL8113Device_StateAT %I*BOOL8116"}
{attribute addProperty CRC "878559470"}
{attribute addProperty SizeInBites "16"}
{attribute addProperty SizeInBytes "2"}
TYPE DeviceState_Inputs_Device_345DC0EE :
STRUCT
	{attribute addProperty Name "Device_Diag"}
	Device_Diag AT %I* : BOOL;
	{attribute addProperty Name "Device_State"}
	Device_State AT %I* : BOOL;
END_STRUCT
END_TYPE

// ---- DUTs/IO/PDOs/DeviceState_Inputs_BDC6BEC3.TcDUT
{attribute addProperty BoxType "EJ6224-0000-0016"}
{attribute addProperty Id "State_Ch1AT %I*USINT811State_Ch2AT %I*USINT812State_Ch3AT %I*USINT813State_Ch4AT %I*USINT814"}
{attribute addProperty CRC "3183918787"}
{attribute addProperty SizeInBites "32"}
{attribute addProperty SizeInBytes "4"}
TYPE DeviceState_Inputs_BDC6BEC3 :
STRUCT
	{attribute addProperty Name "State_Ch1"}
	State_Ch1 AT %I* : USINT;
	{attribute addProperty Name "State_Ch2"}
	State_Ch2 AT %I* : USINT;
	{attribute addProperty Name "State_Ch3"}
	State_Ch3 AT %I* : USINT;
	{attribute addProperty Name "State_Ch4"}
	State_Ch4 AT %I* : USINT;
END_STRUCT
END_TYPE

// ---- DUTs/IO/PDOs/InfoData_275E3363.TcDUT
{attribute addProperty BoxType "EJ6224-0000-0016"}
{attribute addProperty Id "AdsAddrAT %I*AMSADDR6480AoeNetIdAT %I*AMSNETID4860StateAT %I*UINT1620"}
{attribute addProperty CRC "660484963"}
{attribute addProperty SizeInBites "128"}
{attribute addProperty SizeInBytes "16"}
TYPE InfoData_275E3363 :
STRUCT
	{attribute addProperty Name "AdsAddr"}
	AdsAddr AT %I* : AMSADDR;
	{attribute addProperty Name "AoeNetId"}
	AoeNetId AT %I* : AMSNETID;
	{attribute addProperty Name "State"}
	State AT %I* : UINT;
END_STRUCT
END_TYPE

// ---- DUTs/IO/PDOs/Module_1_DeviceState_Inputs_Device_50DD3C95.TcDUT
{attribute addProperty BoxType "EJ6224-0000-0016"}
{attribute addProperty Id "DeviceState_Inputs_DeviceDeviceState_Inputs_Device_345DC0EE162"}
{attribute addProperty CRC "1356676245"}
{attribute addProperty SizeInBites "16"}
{attribute addProperty SizeInBytes "2"}
TYPE Module_1_DeviceState_Inputs_Device_50DD3C95 :
STRUCT
	{attribute addProperty Name "DeviceState_Inputs_Device"}
	DeviceState_Inputs_Device  : DeviceState_Inputs_Device_345DC0EE;
END_STRUCT
END_TYPE

// ---- DUTs/IO/PDOs/Module_2_DeviceState_Inputs_D860B2E3.TcDUT
{attribute addProperty BoxType "EJ6224-0000-0016"}
{attribute addProperty Id "DeviceState_InputsDeviceState_Inputs_BDC6BEC3324"}
{attribute addProperty CRC "3630215907"}
{attribute addProperty SizeInBites "32"}
{attribute addProperty SizeInBytes "4"}
TYPE Module_2_DeviceState_Inputs_D860B2E3 :
STRUCT
	{attribute addProperty Name "DeviceState_Inputs"}
	DeviceState_Inputs  : DeviceState_Inputs_BDC6BEC3;
END_STRUCT
END_TYPE

// ---- DUTs/IO/PDOs/STM_Status_64D93743.TcDUT
{attribute addProperty BoxType "EJ7031-0000-0026"}
{attribute addProperty Id "StatusAT %I*Status_06A4ECA2162"}
{attribute addProperty CRC "1691957059"}
{attribute addProperty SizeInBites "16"}
{attribute addProperty SizeInBytes "2"}
TYPE STM_Status_64D93743 :
STRUCT
	{attribute addProperty Name "Status"}
	Status AT %I* : Status_06A4ECA2;
END_STRUCT
END_TYPE

// ---- DUTs/IO/PDOs/STM_Control_6F24B2C4.TcDUT
{attribute addProperty BoxType "EJ7031-0000-0026"}
{attribute addProperty Id "ControlAT %Q*Control_197B7E66162"}
{attribute addProperty CRC "1864676036"}
{attribute addProperty SizeInBites "16"}
{attribute addProperty SizeInBytes "2"}
TYPE STM_Control_6F24B2C4 :
STRUCT
	{attribute addProperty Name "Control"}
	Control AT %Q* : Control_197B7E66;
END_STRUCT
END_TYPE

// ---- DUTs/IO/PDOs/STM_Velocity_1D89B5C2.TcDUT
{attribute addProperty BoxType "EJ7031-0000-0026"}
{attribute addProperty Id "VelocityAT %Q*INT162"}
{attribute addProperty CRC "495564226"}
{attribute addProperty SizeInBites "16"}
{attribute addProperty SizeInBytes "2"}
TYPE STM_Velocity_1D89B5C2 :
STRUCT
	{attribute addProperty Name "Velocity"}
	Velocity AT %Q* : INT;
END_STRUCT
END_TYPE

// ---- DUTs/IO/PDOs/InfoData_1C46E3E7.TcDUT
{attribute addProperty BoxType "EJ7031-0000-0026"}
{attribute addProperty Id "AdsAddrAT %I*AMSADDR6480Chn0AT %I*USINT810Chn1AT %I*USINT810StateAT %I*UINT1620"}
{attribute addProperty CRC "474407911"}
{attribute addProperty SizeInBites "96"}
{attribute addProperty SizeInBytes "12"}
TYPE InfoData_1C46E3E7 :
STRUCT
	{attribute addProperty Name "AdsAddr"}
	AdsAddr AT %I* : AMSADDR;
	{attribute addProperty Name "Chn0"}
	Chn0 AT %I* : USINT;
	{attribute addProperty Name "Chn1"}
	Chn1 AT %I* : USINT;
	{attribute addProperty Name "State"}
	State AT %I* : UINT;
END_STRUCT
END_TYPE

// ---- DUTs/IO/PDOs/ENC_Status_compact_DA87336C.TcDUT
{attribute addProperty BoxType "EJ7037-0000-0020"}
{attribute addProperty Id "StatusAT %I*Status_E26627ED1621Counter_valueAT %I*UINT16217Latch_valueAT %I*UINT16218"}
{attribute addProperty CRC "3666293612"}
{attribute addProperty SizeInBites "48"}
{attribute addProperty SizeInBytes "6"}
TYPE ENC_Status_compact_DA87336C :
STRUCT
	{attribute addProperty Name "Status"}
	Status AT %I* : Status_E26627ED;
	{attribute addProperty Name "Counter_value"}
	Counter_value AT %I* : UINT;
	{attribute addProperty Name "Latch_value"}
	Latch_value AT %I* : UINT;
END_STRUCT
END_TYPE

// ---- DUTs/IO/PDOs/STM_Status_CB86BB9A.TcDUT
{attribute addProperty BoxType "EJ7037-0000-0020"}
{attribute addProperty Id "StatusAT %I*Status_4F9ADA1B162"}
{attribute addProperty CRC "3414604698"}
{attribute addProperty SizeInBites "16"}
{attribute addProperty SizeInBytes "2"}
TYPE STM_Status_CB86BB9A :
STRUCT
	{attribute addProperty Name "Status"}
	Status AT %I* : Status_4F9ADA1B;
END_STRUCT
END_TYPE

// ---- DUTs/IO/PDOs/STM_Control_91ECC2DE.TcDUT
{attribute addProperty BoxType "EJ7037-0000-0020"}
{attribute addProperty Id "ControlAT %Q*Control_D763B957162"}
{attribute addProperty CRC "2448212702"}
{attribute addProperty SizeInBites "16"}
{attribute addProperty SizeInBytes "2"}
TYPE STM_Control_91ECC2DE :
STRUCT
	{attribute addProperty Name "Control"}
	Control AT %Q* : Control_D763B957;
END_STRUCT
END_TYPE

// ---- DUTs/IO/PDOs/ENC_Status_compact_Channel_559DED98.TcDUT
{attribute addProperty BoxType "EJ7342-0000-0019"}
{attribute addProperty Id "StatusAT %I*Status_4B9F49E31620Counter_valueAT %I*UINT16217Latch_valueAT %I*UINT16218"}
{attribute addProperty CRC "1436413336"}
{attribute addProperty SizeInBites "48"}
{attribute addProperty SizeInBytes "6"}
TYPE ENC_Status_compact_Channel_559DED98 :
STRUCT
	{attribute addProperty Name "Status"}
	Status AT %I* : Status_4B9F49E3;
	{attribute addProperty Name "Counter_value"}
	Counter_value AT %I* : UINT;
	{attribute addProperty Name "Latch_value"}
	Latch_value AT %I* : UINT;
END_STRUCT
END_TYPE

// ---- DUTs/IO/PDOs/DCM_Status_Channel_C2B0CAE1.TcDUT
{attribute addProperty BoxType "EJ7342-0000-0019"}
{attribute addProperty Id "StatusAT %I*Status_1C57BC2B162"}
{attribute addProperty CRC "3266366177"}
{attribute addProperty SizeInBites "16"}
{attribute addProperty SizeInBytes "2"}
TYPE DCM_Status_Channel_C2B0CAE1 :
STRUCT
	{attribute addProperty Name "Status"}
	Status AT %I* : Status_1C57BC2B;
END_STRUCT
END_TYPE

// ---- DUTs/IO/PDOs/ENC_Control_compact_Channel_5C86AA9D.TcDUT
{attribute addProperty BoxType "EJ7342-0000-0019"}
{attribute addProperty Id "ControlAT %Q*Control_E8AFF3DF1620Set_counter_valueAT %Q*UINT16217"}
{attribute addProperty CRC "1552329373"}
{attribute addProperty SizeInBites "32"}
{attribute addProperty SizeInBytes "4"}
TYPE ENC_Control_compact_Channel_5C86AA9D :
STRUCT
	{attribute addProperty Name "Control"}
	Control AT %Q* : Control_E8AFF3DF;
	{attribute addProperty Name "Set_counter_value"}
	Set_counter_value AT %Q* : UINT;
END_STRUCT
END_TYPE

// ---- DUTs/IO/PDOs/DCM_Control_Channel_6F24B2C4.TcDUT
{attribute addProperty BoxType "EJ7342-0000-0019"}
{attribute addProperty Id "ControlAT %Q*Control_197B7E66162"}
{attribute addProperty CRC "1864676036"}
{attribute addProperty SizeInBites "16"}
{attribute addProperty SizeInBytes "2"}
TYPE DCM_Control_Channel_6F24B2C4 :
STRUCT
	{attribute addProperty Name "Control"}
	Control AT %Q* : Control_197B7E66;
END_STRUCT
END_TYPE

// ---- DUTs/IO/PDOs/DCM_Velocity_Channel_1D89B5C2.TcDUT
{attribute addProperty BoxType "EJ7342-0000-0019"}
{attribute addProperty Id "VelocityAT %Q*INT162"}
{attribute addProperty CRC "495564226"}
{attribute addProperty SizeInBites "16"}
{attribute addProperty SizeInBytes "2"}
TYPE DCM_Velocity_Channel_1D89B5C2 :
STRUCT
	{attribute addProperty Name "Velocity"}
	Velocity AT %Q* : INT;
END_STRUCT
END_TYPE

// ---- DUTs/IO/PDOs/InfoData_3F3BB279.TcDUT
{attribute addProperty BoxType "EJ7342-0000-0019"}
{attribute addProperty Id "AdsAddrAT %I*AMSADDR6480Chn0AT %I*USINT810Chn1AT %I*USINT810Chn2AT %I*USINT810Chn3AT %I*USINT810StateAT %I*UINT1620"}
{attribute addProperty CRC "1060876921"}
{attribute addProperty SizeInBites "112"}
{attribute addProperty SizeInBytes "14"}
TYPE InfoData_3F3BB279 :
STRUCT
	{attribute addProperty Name "AdsAddr"}
	AdsAddr AT %I* : AMSADDR;
	{attribute addProperty Name "Chn0"}
	Chn0 AT %I* : USINT;
	{attribute addProperty Name "Chn1"}
	Chn1 AT %I* : USINT;
	{attribute addProperty Name "Chn2"}
	Chn2 AT %I* : USINT;
	{attribute addProperty Name "Chn3"}
	Chn3 AT %I* : USINT;
	{attribute addProperty Name "State"}
	State AT %I* : UINT;
END_STRUCT
END_TYPE

// ---- DUTs/IO/PDOs/ENC_Status_compact_Channel_A7E8355C.TcDUT
{attribute addProperty BoxType "EJ7342-0000-0020"}
{attribute addProperty Id "StatusAT %I*Status_A881DFA01620Counter_valueAT %I*UINT16217Latch_valueAT %I*UINT16218"}
{attribute addProperty CRC "2817013084"}
{attribute addProperty SizeInBites "48"}
{attribute addProperty SizeInBytes "6"}
TYPE ENC_Status_compact_Channel_A7E8355C :
STRUCT
	{attribute addProperty Name "Status"}
	Status AT %I* : Status_A881DFA0;
	{attribute addProperty Name "Counter_value"}
	Counter_value AT %I* : UINT;
	{attribute addProperty Name "Latch_value"}
	Latch_value AT %I* : UINT;
END_STRUCT
END_TYPE

// ---- DUTs/IO/PDOs/DCM_Status_Channel_64D93743.TcDUT
{attribute addProperty BoxType "EJ7342-0000-0020"}
{attribute addProperty Id "StatusAT %I*Status_06A4ECA2162"}
{attribute addProperty CRC "1691957059"}
{attribute addProperty SizeInBites "16"}
{attribute addProperty SizeInBytes "2"}
TYPE DCM_Status_Channel_64D93743 :
STRUCT
	{attribute addProperty Name "Status"}
	Status AT %I* : Status_06A4ECA2;
END_STRUCT
END_TYPE

// ---- DUTs/IO/PDOs/FB_Position_BA8AA9F0.TcDUT
{attribute addProperty BoxType "EJ7211-0010-0026"}
{attribute addProperty Id "PositionAT %I*UDINT324"}
{attribute addProperty CRC "3129649648"}
{attribute addProperty SizeInBites "32"}
{attribute addProperty SizeInBytes "4"}
TYPE FB_Position_BA8AA9F0 :
STRUCT
	{attribute addProperty Name "Position"}
	Position AT %I* : UDINT;
END_STRUCT
END_TYPE

// ---- DUTs/IO/PDOs/DRV_Statusword_53CBCECC.TcDUT
{attribute addProperty BoxType "EJ7211-0010-0026"}
{attribute addProperty Id "StatuswordAT %I*UINT162"}
{attribute addProperty CRC "1405865676"}
{attribute addProperty SizeInBites "16"}
{attribute addProperty SizeInBytes "2"}
TYPE DRV_Statusword_53CBCECC :
STRUCT
	{attribute addProperty Name "Statusword"}
	Statusword AT %I* : UINT;
END_STRUCT
END_TYPE

// ---- DUTs/IO/PDOs/DRV_Controlword_41761768.TcDUT
{attribute addProperty BoxType "EJ7211-0010-0026"}
{attribute addProperty Id "ControlwordAT %Q*UINT162"}
{attribute addProperty CRC "1098258280"}
{attribute addProperty SizeInBites "16"}
{attribute addProperty SizeInBytes "2"}
TYPE DRV_Controlword_41761768 :
STRUCT
	{attribute addProperty Name "Controlword"}
	Controlword AT %Q* : UINT;
END_STRUCT
END_TYPE

// ---- DUTs/IO/PDOs/DRV_Target_velocity_53A88AB0.TcDUT
{attribute addProperty BoxType "EJ7211-0010-0026"}
{attribute addProperty Id "Target_velocityAT %Q*DINT324"}
{attribute addProperty CRC "1403554480"}
{attribute addProperty SizeInBites "32"}
{attribute addProperty SizeInBytes "4"}
TYPE DRV_Target_velocity_53A88AB0 :
STRUCT
	{attribute addProperty Name "Target_velocity"}
	Target_velocity AT %Q* : DINT;
END_STRUCT
END_TYPE

// ---- DUTs/IO/PDOs/InfoData_AEB17F4D.TcDUT
{attribute addProperty BoxType "EJ7211-0010-0026"}
{attribute addProperty Id "AdsAddrAT %I*AMSADDR6480DcOutputShiftAT %I*DINT3240DcInputShiftAT %I*DINT3240Chn0AT %I*USINT810StateAT %I*UINT1620"}
{attribute addProperty CRC "2930868045"}
{attribute addProperty SizeInBites "152"}
{attribute addProperty SizeInBytes "19"}
TYPE InfoData_AEB17F4D :
STRUCT
	{attribute addProperty Name "AdsAddr"}
	AdsAddr AT %I* : AMSADDR;
	{attribute addProperty Name "DcOutputShift"}
	DcOutputShift AT %I* : DINT;
	{attribute addProperty Name "DcInputShift"}
	DcInputShift AT %I* : DINT;
	{attribute addProperty Name "Chn0"}
	Chn0 AT %I* : USINT;
	{attribute addProperty Name "State"}
	State AT %I* : UINT;
END_STRUCT
END_TYPE

// ---- DUTs/IO/PDOs/InfoData_81099714.TcDUT
{attribute addProperty BoxType "EJ7211-0010-0030"}
{attribute addProperty Id "AdsAddrAT %I*AMSADDR6480DcOutputShiftAT %I*DINT3240DcInputShiftAT %I*DINT3240Chn0AT %I*USINT810Chn1AT %I*USINT810StateAT %I*UINT1620"}
{attribute addProperty CRC "2164889364"}
{attribute addProperty SizeInBites "160"}
{attribute addProperty SizeInBytes "20"}
TYPE InfoData_81099714 :
STRUCT
	{attribute addProperty Name "AdsAddr"}
	AdsAddr AT %I* : AMSADDR;
	{attribute addProperty Name "DcOutputShift"}
	DcOutputShift AT %I* : DINT;
	{attribute addProperty Name "DcInputShift"}
	DcInputShift AT %I* : DINT;
	{attribute addProperty Name "Chn0"}
	Chn0 AT %I* : USINT;
	{attribute addProperty Name "Chn1"}
	Chn1 AT %I* : USINT;
	{attribute addProperty Name "State"}
	State AT %I* : UINT;
END_STRUCT
END_TYPE

// ---- DUTs/IO/PDOs/DS402_Statusword_53CBCECC.TcDUT
{attribute addProperty BoxType "EJ7211-0011-0026"}
{attribute addProperty Id "StatuswordAT %I*UINT162"}
{attribute addProperty CRC "1405865676"}
{attribute addProperty SizeInBites "16"}
{attribute addProperty SizeInBytes "2"}
TYPE DS402_Statusword_53CBCECC :
STRUCT
	{attribute addProperty Name "Statusword"}
	Statusword AT %I* : UINT;
END_STRUCT
END_TYPE

// ---- DUTs/IO/PDOs/DS402_Position_actual_value_0D11C114.TcDUT
{attribute addProperty BoxType "EJ7211-0011-0026"}
{attribute addProperty Id "Position_actual_valueAT %I*UDINT324"}
{attribute addProperty CRC "219267348"}
{attribute addProperty SizeInBites "32"}
{attribute addProperty SizeInBytes "4"}
TYPE DS402_Position_actual_value_0D11C114 :
STRUCT
	{attribute addProperty Name "Position_actual_value"}
	Position_actual_value AT %I* : UDINT;
END_STRUCT
END_TYPE

// ---- DUTs/IO/PDOs/DS402_Controlword_41761768.TcDUT
{attribute addProperty BoxType "EJ7211-0011-0026"}
{attribute addProperty Id "ControlwordAT %Q*UINT162"}
{attribute addProperty CRC "1098258280"}
{attribute addProperty SizeInBites "16"}
{attribute addProperty SizeInBytes "2"}
TYPE DS402_Controlword_41761768 :
STRUCT
	{attribute addProperty Name "Controlword"}
	Controlword AT %Q* : UINT;
END_STRUCT
END_TYPE

// ---- DUTs/IO/PDOs/DS402_Target_velocity_53A88AB0.TcDUT
{attribute addProperty BoxType "EJ7211-0011-0026"}
{attribute addProperty Id "Target_velocityAT %Q*DINT324"}
{attribute addProperty CRC "1403554480"}
{attribute addProperty SizeInBites "32"}
{attribute addProperty SizeInBytes "4"}
TYPE DS402_Target_velocity_53A88AB0 :
STRUCT
	{attribute addProperty Name "Target_velocity"}
	Target_velocity AT %Q* : DINT;
END_STRUCT
END_TYPE

// ---- DUTs/IO/PDOs/InfoData_BF6E01EA.TcDUT
{attribute addProperty BoxType "EJ7211-9414-0030"}
{attribute addProperty Id "AdsAddrAT %I*AMSADDR6480DcOutputShiftAT %I*DINT3240DcInputShiftAT %I*DINT3240Chn0AT %I*USINT810Chn1AT %I*USINT810Chn2AT %I*USINT810StateAT %I*UINT1620"}
{attribute addProperty CRC "3211657706"}
{attribute addProperty SizeInBites "168"}
{attribute addProperty SizeInBytes "21"}
TYPE InfoData_BF6E01EA :
STRUCT
	{attribute addProperty Name "AdsAddr"}
	AdsAddr AT %I* : AMSADDR;
	{attribute addProperty Name "DcOutputShift"}
	DcOutputShift AT %I* : DINT;
	{attribute addProperty Name "DcInputShift"}
	DcInputShift AT %I* : DINT;
	{attribute addProperty Name "Chn0"}
	Chn0 AT %I* : USINT;
	{attribute addProperty Name "Chn1"}
	Chn1 AT %I* : USINT;
	{attribute addProperty Name "Chn2"}
	Chn2 AT %I* : USINT;
	{attribute addProperty Name "State"}
	State AT %I* : UINT;
END_STRUCT
END_TYPE

// ---- DUTs/IO/PDOs/DCM_Status_Channel_DBE0EA1F.TcDUT
{attribute addProperty BoxType "EJ7334-0008-0016"}
{attribute addProperty Id "StatusAT %I*Status_7570E3BD162"}
{attribute addProperty CRC "3688950303"}
{attribute addProperty SizeInBites "16"}
{attribute addProperty SizeInBytes "2"}
TYPE DCM_Status_Channel_DBE0EA1F :
STRUCT
	{attribute addProperty Name "Status"}
	Status AT %I* : Status_7570E3BD;
END_STRUCT
END_TYPE

// ---- DUTs/IO/PDOs/DCM_Outputs_Channel_1F77C8C2.TcDUT
{attribute addProperty BoxType "EJ7334-0008-0016"}
{attribute addProperty Id "ControlAT %Q*Control_96E4A9881621VelocityAT %Q*INT16233"}
{attribute addProperty CRC "527943874"}
{attribute addProperty SizeInBites "32"}
{attribute addProperty SizeInBytes "4"}
TYPE DCM_Outputs_Channel_1F77C8C2 :
STRUCT
	{attribute addProperty Name "Control"}
	Control AT %Q* : Control_96E4A988;
	{attribute addProperty Name "Velocity"}
	Velocity AT %Q* : INT;
END_STRUCT
END_TYPE

// ---- DUTs/IO/PDOs/DRV_Following_error_actual_value_F5433536.TcDUT
{attribute addProperty BoxType "EJ7411-0000-0018"}
{attribute addProperty Id "Following_error_actual_valueAT %I*DINT324"}
{attribute addProperty CRC "4114822454"}
{attribute addProperty SizeInBites "32"}
{attribute addProperty SizeInBytes "4"}
TYPE DRV_Following_error_actual_value_F5433536 :
STRUCT
	{attribute addProperty Name "Following_error_actual_value"}
	Following_error_actual_value AT %I* : DINT;
END_STRUCT
END_TYPE

// ---- DUTs/IO/PDOs/DRV_Target_position_41334FAA.TcDUT
{attribute addProperty BoxType "EJ7411-0000-0018"}
{attribute addProperty Id "Target_positionAT %Q*UDINT324"}
{attribute addProperty CRC "1093881770"}
{attribute addProperty SizeInBites "32"}
{attribute addProperty SizeInBytes "4"}
TYPE DRV_Target_position_41334FAA :
STRUCT
	{attribute addProperty Name "Target_position"}
	Target_position AT %Q* : UDINT;
END_STRUCT
END_TYPE

// ---- DUTs/IO/PDOs/Status_Uo_D2430366.TcDUT
{attribute addProperty BoxType "EJ9505-0000-0016"}
{attribute addProperty Id "Power_OKAT %I*BOOL811OverloadAT %I*BOOL812"}
{attribute addProperty CRC "3527607142"}
{attribute addProperty SizeInBites "16"}
{attribute addProperty SizeInBytes "2"}
TYPE Status_Uo_D2430366 :
STRUCT
	{attribute addProperty Name "Power_OK"}
	Power_OK AT %I* : BOOL;
	{attribute addProperty Name "Overload"}
	Overload AT %I* : BOOL;
END_STRUCT
END_TYPE

// ---- DUTs/IO/PDOs/BCT_Inputs_7F924099.TcDUT
{attribute addProperty BoxType "EJ9576-0000-0018"}
{attribute addProperty Id "Terminal_OvertemperatureAT %I*BOOL811I2T_errorAT %I*BOOL812I2T_warningAT %I*BOOL813OvervoltageAT %I*BOOL814UndervoltageAT %I*BOOL815Chopper_onAT %I*BOOL816Input_cycle_counterAT %I*BYTE8115DC_link_voltageAT %I*UDINT32417Resistor_currentAT %I*DINT32419Duty_cylceAT %I*USINT8120"}
{attribute addProperty CRC "2140291225"}
{attribute addProperty SizeInBites "128"}
{attribute addProperty SizeInBytes "16"}
TYPE BCT_Inputs_7F924099 :
STRUCT
	{attribute addProperty Name "Terminal_Overtemperature"}
	Terminal_Overtemperature AT %I* : BOOL;
	{attribute addProperty Name "I2T_error"}
	I2T_error AT %I* : BOOL;
	{attribute addProperty Name "I2T_warning"}
	I2T_warning AT %I* : BOOL;
	{attribute addProperty Name "Overvoltage"}
	Overvoltage AT %I* : BOOL;
	{attribute addProperty Name "Undervoltage"}
	Undervoltage AT %I* : BOOL;
	{attribute addProperty Name "Chopper_on"}
	Chopper_on AT %I* : BOOL;
	{attribute addProperty Name "Input_cycle_counter"}
	Input_cycle_counter AT %I* : BYTE;
	{attribute addProperty Name "DC_link_voltage"}
	DC_link_voltage AT %I* : UDINT;
	{attribute addProperty Name "Resistor_current"}
	Resistor_current AT %I* : DINT;
	{attribute addProperty Name "Duty_cylce"}
	Duty_cylce AT %I* : USINT;
END_STRUCT
END_TYPE

// ---- DUTs/IO/PDOs/BCT_Inputs_6A3D8194.TcDUT
{attribute addProperty BoxType "EJ9576-0000-0019"}
{attribute addProperty Id "Terminal_OvertemperatureAT %I*BOOL811I2T_errorAT %I*BOOL812I2T_warningAT %I*BOOL813OvervoltageAT %I*BOOL814UndervoltageAT %I*BOOL815Chopper_onAT %I*BOOL816Input_cycle_counterAT %I*BYTE8115DC_link_voltageAT %I*UDINT32417Resistor_currentAT %I*DINT32419Duty_cylceAT %I*USINT8120I2T_load_factorAT %I*USINT8121"}
{attribute addProperty CRC "1782415764"}
{attribute addProperty SizeInBites "136"}
{attribute addProperty SizeInBytes "17"}
TYPE BCT_Inputs_6A3D8194 :
STRUCT
	{attribute addProperty Name "Terminal_Overtemperature"}
	Terminal_Overtemperature AT %I* : BOOL;
	{attribute addProperty Name "I2T_error"}
	I2T_error AT %I* : BOOL;
	{attribute addProperty Name "I2T_warning"}
	I2T_warning AT %I* : BOOL;
	{attribute addProperty Name "Overvoltage"}
	Overvoltage AT %I* : BOOL;
	{attribute addProperty Name "Undervoltage"}
	Undervoltage AT %I* : BOOL;
	{attribute addProperty Name "Chopper_on"}
	Chopper_on AT %I* : BOOL;
	{attribute addProperty Name "Input_cycle_counter"}
	Input_cycle_counter AT %I* : BYTE;
	{attribute addProperty Name "DC_link_voltage"}
	DC_link_voltage AT %I* : UDINT;
	{attribute addProperty Name "Resistor_current"}
	Resistor_current AT %I* : DINT;
	{attribute addProperty Name "Duty_cylce"}
	Duty_cylce AT %I* : USINT;
	{attribute addProperty Name "I2T_load_factor"}
	I2T_load_factor AT %I* : USINT;
END_STRUCT
END_TYPE

// ---- DUTs/IO/PDOs/BCT_Inputs_047F8208.TcDUT
{attribute addProperty BoxType "EJ9576-0000-0020"}
{attribute addProperty Id "Terminal_OvertemperatureAT %I*BOOL811I2T_errorAT %I*BOOL812I2T_warningAT %I*BOOL813OvervoltageAT %I*BOOL814UndervoltageAT %I*BOOL815Chopper_onAT %I*BOOL816Input_cycle_counterAT %I*BYTE8115DC_link_voltageAT %I*UDINT32417Resistor_CurrentAT %I*DINT32419Duty_CycleAT %I*USINT8120"}
{attribute addProperty CRC "75465224"}
{attribute addProperty SizeInBites "128"}
{attribute addProperty SizeInBytes "16"}
TYPE BCT_Inputs_047F8208 :
STRUCT
	{attribute addProperty Name "Terminal_Overtemperature"}
	Terminal_Overtemperature AT %I* : BOOL;
	{attribute addProperty Name "I2T_error"}
	I2T_error AT %I* : BOOL;
	{attribute addProperty Name "I2T_warning"}
	I2T_warning AT %I* : BOOL;
	{attribute addProperty Name "Overvoltage"}
	Overvoltage AT %I* : BOOL;
	{attribute addProperty Name "Undervoltage"}
	Undervoltage AT %I* : BOOL;
	{attribute addProperty Name "Chopper_on"}
	Chopper_on AT %I* : BOOL;
	{attribute addProperty Name "Input_cycle_counter"}
	Input_cycle_counter AT %I* : BYTE;
	{attribute addProperty Name "DC_link_voltage"}
	DC_link_voltage AT %I* : UDINT;
	{attribute addProperty Name "Resistor_Current"}
	Resistor_Current AT %I* : DINT;
	{attribute addProperty Name "Duty_Cycle"}
	Duty_Cycle AT %I* : USINT;
END_STRUCT
END_TYPE

// ---- DUTs/IO/PDOs/BCT_Inputs_4FFA390D.TcDUT
{attribute addProperty BoxType "EJ9576-0000-0022"}
{attribute addProperty Id "Terminal_OvertemperatureAT %I*BOOL811I2T_errorAT %I*BOOL812I2T_warningAT %I*BOOL813OvervoltageAT %I*BOOL814UndervoltageAT %I*BOOL815Chopper_onAT %I*BOOL816Overcurrent_ProtectionAT %I*BOOL817Input_cycle_counterAT %I*BYTE8115DC_link_voltageAT %I*UDINT32417Resistor_CurrentAT %I*DINT32419Duty_CycleAT %I*USINT8120"}
{attribute addProperty CRC "1341798669"}
{attribute addProperty SizeInBites "136"}
{attribute addProperty SizeInBytes "17"}
TYPE BCT_Inputs_4FFA390D :
STRUCT
	{attribute addProperty Name "Terminal_Overtemperature"}
	Terminal_Overtemperature AT %I* : BOOL;
	{attribute addProperty Name "I2T_error"}
	I2T_error AT %I* : BOOL;
	{attribute addProperty Name "I2T_warning"}
	I2T_warning AT %I* : BOOL;
	{attribute addProperty Name "Overvoltage"}
	Overvoltage AT %I* : BOOL;
	{attribute addProperty Name "Undervoltage"}
	Undervoltage AT %I* : BOOL;
	{attribute addProperty Name "Chopper_on"}
	Chopper_on AT %I* : BOOL;
	{attribute addProperty Name "Overcurrent_Protection"}
	Overcurrent_Protection AT %I* : BOOL;
	{attribute addProperty Name "Input_cycle_counter"}
	Input_cycle_counter AT %I* : BYTE;
	{attribute addProperty Name "DC_link_voltage"}
	DC_link_voltage AT %I* : UDINT;
	{attribute addProperty Name "Resistor_Current"}
	Resistor_Current AT %I* : DINT;
	{attribute addProperty Name "Duty_Cycle"}
	Duty_Cycle AT %I* : USINT;
END_STRUCT
END_TYPE

// ---- DUTs/IO/PDOs/FSoE_Inputs_899BAC0E.TcDUT
{attribute addProperty BoxType "EJ1914-0000-0017"}
{attribute addProperty Id "FSOEAT %I*FSOE_4B534C96486"}
{attribute addProperty CRC "2308680718"}
{attribute addProperty SizeInBites "48"}
{attribute addProperty SizeInBytes "6"}
TYPE FSoE_Inputs_899BAC0E :
STRUCT
	{attribute addProperty Name "FSOE"}
	FSOE AT %I* : FSOE_4B534C96;
END_STRUCT
END_TYPE

// ---- DUTs/IO/PDOs/FSoE_Outputs_E28701A0.TcDUT
{attribute addProperty BoxType "EJ1914-0000-0017"}
{attribute addProperty Id "FSOEAT %Q*FSOE_27E40C71486"}
{attribute addProperty CRC "3800498592"}
{attribute addProperty SizeInBites "48"}
{attribute addProperty SizeInBytes "6"}
TYPE FSoE_Outputs_E28701A0 :
STRUCT
	{attribute addProperty Name "FSOE"}
	FSOE AT %Q* : FSOE_27E40C71;
END_STRUCT
END_TYPE

// ---- DUTs/IO/PDOs/FIELDVOLTAGE_Field_Voltage_Status_CAC01FE2.TcDUT
{attribute addProperty BoxType "EJ1914-0000-0017"}
{attribute addProperty Id "Fieldvoltage_UnderrangeAT %I*BOOL811Fieldvoltage_OverrangeAT %I*BOOL812"}
{attribute addProperty CRC "3401588706"}
{attribute addProperty SizeInBites "16"}
{attribute addProperty SizeInBytes "2"}
TYPE FIELDVOLTAGE_Field_Voltage_Status_CAC01FE2 :
STRUCT
	{attribute addProperty Name "Fieldvoltage_Underrange"}
	Fieldvoltage_Underrange AT %I* : BOOL;
	{attribute addProperty Name "Fieldvoltage_Overrange"}
	Fieldvoltage_Overrange AT %I* : BOOL;
END_STRUCT
END_TYPE

// ---- DUTs/IO/PDOs/FSLOGIC_Inputs_8BA5C933.TcDUT
{attribute addProperty BoxType "EJ1914-0000-0017"}
{attribute addProperty Id "Safe_Logic_StateAT %I*USINT811Cycle_CounterAT %I*USINT812"}
{attribute addProperty CRC "2342897971"}
{attribute addProperty SizeInBites "16"}
{attribute addProperty SizeInBytes "2"}
TYPE FSLOGIC_Inputs_8BA5C933 :
STRUCT
	{attribute addProperty Name "Safe_Logic_State"}
	Safe_Logic_State AT %I* : USINT;
	{attribute addProperty Name "Cycle_Counter"}
	Cycle_Counter AT %I* : USINT;
END_STRUCT
END_TYPE

// ---- DUTs/IO/PDOs/EMPTY_STRUCTURE.TcDUT
{attribute addProperty BoxType "EJ1914-0000-0017"}
{attribute addProperty Id "EMPTY_STRUCTURE"}
{attribute addProperty CRC "0"}
{attribute addProperty SizeInBites "0"}
{attribute addProperty SizeInBytes "0"}
TYPE EMPTY_STRUCTURE :
STRUCT
END_STRUCT
END_TYPE

// ---- DUTs/IO/PDOs/Module_1_FSOE_60919941.TcDUT
{attribute addProperty BoxType "EJ1914-0000-0017"}
{attribute addProperty Id "FSoE_InputsFSoE_Inputs_899BAC0E486FSoE_OutputsFSoE_Outputs_E28701A0486"}
{attribute addProperty CRC "1620154689"}
{attribute addProperty SizeInBites "96"}
{attribute addProperty SizeInBytes "12"}
TYPE Module_1_FSOE_60919941 :
STRUCT
	{attribute addProperty Name "FSoE_Inputs"}
	FSoE_Inputs  : FSoE_Inputs_899BAC0E;
	{attribute addProperty Name "FSoE_Outputs"}
	FSoE_Outputs  : FSoE_Outputs_E28701A0;
END_STRUCT
END_TYPE

// ---- DUTs/IO/PDOs/Module_2_DEVICEIO_FB2B67D7.TcDUT
{attribute addProperty BoxType "EJ1914-0000-0017"}
{attribute addProperty Id "FIELDVOLTAGE_Field_Voltage_StatusFIELDVOLTAGE_Field_Voltage_Status_CAC01FE2162"}
{attribute addProperty CRC "4213925847"}
{attribute addProperty SizeInBites "16"}
{attribute addProperty SizeInBytes "2"}
TYPE Module_2_DEVICEIO_FB2B67D7 :
STRUCT
	{attribute addProperty Name "FIELDVOLTAGE_Field_Voltage_Status"}
	FIELDVOLTAGE_Field_Voltage_Status  : FIELDVOLTAGE_Field_Voltage_Status_CAC01FE2;
END_STRUCT
END_TYPE

// ---- DUTs/IO/PDOs/Module_3_FSLOGIC_3E625139.TcDUT
{attribute addProperty BoxType "EJ1914-0000-0017"}
{attribute addProperty Id "FSLOGIC_InputsFSLOGIC_Inputs_8BA5C933162FSLOGIC_OutputsEMPTY_STRUCTURE00"}
{attribute addProperty CRC "1046630713"}
{attribute addProperty SizeInBites "16"}
{attribute addProperty SizeInBytes "2"}
TYPE Module_3_FSLOGIC_3E625139 :
STRUCT
	{attribute addProperty Name "FSLOGIC_Inputs"}
	FSLOGIC_Inputs  : FSLOGIC_Inputs_8BA5C933;
	{attribute addProperty Name "FSLOGIC_Outputs"}
	FSLOGIC_Outputs  : EMPTY_STRUCTURE;
END_STRUCT
END_TYPE

// ---- DUTs/IO/PDOs/FSoE_Inputs_2B542CE7.TcDUT
{attribute addProperty BoxType "EJ1918-0000-0017"}
{attribute addProperty Id "FSOEAT %I*FSOE_314B848F567"}
{attribute addProperty CRC "726936807"}
{attribute addProperty SizeInBites "56"}
{attribute addProperty SizeInBytes "7"}
TYPE FSoE_Inputs_2B542CE7 :
STRUCT
	{attribute addProperty Name "FSOE"}
	FSOE AT %I* : FSOE_314B848F;
END_STRUCT
END_TYPE

// ---- DUTs/IO/PDOs/FSoE_Outputs_F12FD39F.TcDUT
{attribute addProperty BoxType "EJ1918-0000-0017"}
{attribute addProperty Id "FSOEAT %Q*FSOE_F333FD78486"}
{attribute addProperty CRC "4046443423"}
{attribute addProperty SizeInBites "48"}
{attribute addProperty SizeInBytes "6"}
TYPE FSoE_Outputs_F12FD39F :
STRUCT
	{attribute addProperty Name "FSOE"}
	FSOE AT %Q* : FSOE_F333FD78;
END_STRUCT
END_TYPE

// ---- DUTs/IO/PDOs/Module_1_FSOE_99CFC0AE.TcDUT
{attribute addProperty BoxType "EJ1918-0000-0017"}
{attribute addProperty Id "FSoE_InputsFSoE_Inputs_2B542CE7567FSoE_OutputsFSoE_Outputs_F12FD39F486"}
{attribute addProperty CRC "2580529326"}
{attribute addProperty SizeInBites "104"}
{attribute addProperty SizeInBytes "13"}
TYPE Module_1_FSOE_99CFC0AE :
STRUCT
	{attribute addProperty Name "FSoE_Inputs"}
	FSoE_Inputs  : FSoE_Inputs_2B542CE7;
	{attribute addProperty Name "FSoE_Outputs"}
	FSoE_Outputs  : FSoE_Outputs_F12FD39F;
END_STRUCT
END_TYPE

// ---- DUTs/IO/PDOs/FSoE_Inputs_E4152F08.TcDUT
{attribute addProperty BoxType "EJ1957-0000-0017"}
{attribute addProperty Id "FSOEAT %I*FSOE_085426AE567"}
{attribute addProperty CRC "3826593544"}
{attribute addProperty SizeInBites "56"}
{attribute addProperty SizeInBytes "7"}
TYPE FSoE_Inputs_E4152F08 :
STRUCT
	{attribute addProperty Name "FSOE"}
	FSOE AT %I* : FSOE_085426AE;
END_STRUCT
END_TYPE

// ---- DUTs/IO/PDOs/FSoE_Outputs_865CD7FA.TcDUT
{attribute addProperty BoxType "EJ1957-0000-0017"}
{attribute addProperty Id "FSOEAT %Q*FSOE_624AB0F2567"}
{attribute addProperty CRC "2254231546"}
{attribute addProperty SizeInBites "56"}
{attribute addProperty SizeInBytes "7"}
TYPE FSoE_Outputs_865CD7FA :
STRUCT
	{attribute addProperty Name "FSOE"}
	FSOE AT %Q* : FSOE_624AB0F2;
END_STRUCT
END_TYPE

// ---- DUTs/IO/PDOs/Outputs_32B9F5E1.TcDUT
{attribute addProperty BoxType "EJ1957-0000-0017"}
{attribute addProperty Id "Channel_1_Standard_OutputAT %Q*BOOL811Channel_2_Standard_OutputAT %Q*BOOL812Channel_3_Standard_OutputAT %Q*BOOL813Channel_4_Standard_OutputAT %Q*BOOL814"}
{attribute addProperty CRC "851047905"}
{attribute addProperty SizeInBites "32"}
{attribute addProperty SizeInBytes "4"}
TYPE Outputs_32B9F5E1 :
STRUCT
	{attribute addProperty Name "Channel_1_Standard_Output"}
	Channel_1_Standard_Output AT %Q* : BOOL;
	{attribute addProperty Name "Channel_2_Standard_Output"}
	Channel_2_Standard_Output AT %Q* : BOOL;
	{attribute addProperty Name "Channel_3_Standard_Output"}
	Channel_3_Standard_Output AT %Q* : BOOL;
	{attribute addProperty Name "Channel_4_Standard_Output"}
	Channel_4_Standard_Output AT %Q* : BOOL;
END_STRUCT
END_TYPE

// ---- DUTs/IO/PDOs/WcState_DC9C9715.TcDUT
{attribute addProperty BoxType "EJ1957-0000-0017"}
{attribute addProperty Id "WcState0AT %I*BIT10.1250WcState1AT %I*BIT10.1250InputToggle0AT %I*BIT10.1250InputToggle1AT %I*BIT10.1250"}
{attribute addProperty CRC "3701249813"}
{attribute addProperty SizeInBites "4"}
{attribute addProperty SizeInBytes "0.5"}
TYPE WcState_DC9C9715 :
STRUCT
	{attribute addProperty Name "WcState0"}
	WcState0 AT %I* : BOOL;
	{attribute addProperty Name "WcState1"}
	WcState1 AT %I* : BOOL;
	{attribute addProperty Name "InputToggle0"}
	InputToggle0 AT %I* : BOOL;
	{attribute addProperty Name "InputToggle1"}
	InputToggle1 AT %I* : BOOL;
END_STRUCT
END_TYPE

// ---- DUTs/IO/PDOs/Module_1_FSOE_B52BB714.TcDUT
{attribute addProperty BoxType "EJ1957-0000-0017"}
{attribute addProperty Id "FSoE_InputsFSoE_Inputs_E4152F08567FSoE_OutputsFSoE_Outputs_865CD7FA567"}
{attribute addProperty CRC "3039541012"}
{attribute addProperty SizeInBites "112"}
{attribute addProperty SizeInBytes "14"}
TYPE Module_1_FSOE_B52BB714 :
STRUCT
	{attribute addProperty Name "FSoE_Inputs"}
	FSoE_Inputs  : FSoE_Inputs_E4152F08;
	{attribute addProperty Name "FSoE_Outputs"}
	FSoE_Outputs  : FSoE_Outputs_865CD7FA;
END_STRUCT
END_TYPE

// ---- DUTs/IO/PDOs/Module_2_FSOUT_B889B7D0.TcDUT
{attribute addProperty BoxType "EJ1957-0000-0017"}
{attribute addProperty Id "OutputsOutputs_32B9F5E1324"}
{attribute addProperty CRC "3096033232"}
{attribute addProperty SizeInBites "32"}
{attribute addProperty SizeInBytes "4"}
TYPE Module_2_FSOUT_B889B7D0 :
STRUCT
	{attribute addProperty Name "Outputs"}
	Outputs  : Outputs_32B9F5E1;
END_STRUCT
END_TYPE

// ---- DUTs/IO/PDOs/Module_3_DEVICEIO_FB2B67D7.TcDUT
{attribute addProperty BoxType "EJ1957-0000-0017"}
{attribute addProperty Id "FIELDVOLTAGE_Field_Voltage_StatusFIELDVOLTAGE_Field_Voltage_Status_CAC01FE2162"}
{attribute addProperty CRC "4213925847"}
{attribute addProperty SizeInBites "16"}
{attribute addProperty SizeInBytes "2"}
TYPE Module_3_DEVICEIO_FB2B67D7 :
STRUCT
	{attribute addProperty Name "FIELDVOLTAGE_Field_Voltage_Status"}
	FIELDVOLTAGE_Field_Voltage_Status  : FIELDVOLTAGE_Field_Voltage_Status_CAC01FE2;
END_STRUCT
END_TYPE

// ---- DUTs/IO/PDOs/Module_4_FSLOGIC_3E625139.TcDUT
{attribute addProperty BoxType "EJ1957-0000-0017"}
{attribute addProperty Id "FSLOGIC_InputsFSLOGIC_Inputs_8BA5C933162FSLOGIC_OutputsEMPTY_STRUCTURE00"}
{attribute addProperty CRC "1046630713"}
{attribute addProperty SizeInBites "16"}
{attribute addProperty SizeInBytes "2"}
TYPE Module_4_FSLOGIC_3E625139 :
STRUCT
	{attribute addProperty Name "FSLOGIC_Inputs"}
	FSLOGIC_Inputs  : FSLOGIC_Inputs_8BA5C933;
	{attribute addProperty Name "FSLOGIC_Outputs"}
	FSLOGIC_Outputs  : EMPTY_STRUCTURE;
END_STRUCT
END_TYPE

// ---- DUTs/IO/PDOs/FSoE_Inputs_74C0DA41.TcDUT
{attribute addProperty BoxType "EJ2914-0000-0017"}
{attribute addProperty Id "FSOEAT %I*FSOE_869360C3486"}
{attribute addProperty CRC "1958795841"}
{attribute addProperty SizeInBites "48"}
{attribute addProperty SizeInBytes "6"}
TYPE FSoE_Inputs_74C0DA41 :
STRUCT
	{attribute addProperty Name "FSOE"}
	FSOE AT %I* : FSOE_869360C3;
END_STRUCT
END_TYPE

// ---- DUTs/IO/PDOs/FSoE_Outputs_841EDA4B.TcDUT
{attribute addProperty BoxType "EJ2914-0000-0017"}
{attribute addProperty Id "FSOEAT %Q*FSOE_108803C1486"}
{attribute addProperty CRC "2216614475"}
{attribute addProperty SizeInBites "48"}
{attribute addProperty SizeInBytes "6"}
TYPE FSoE_Outputs_841EDA4B :
STRUCT
	{attribute addProperty Name "FSOE"}
	FSOE AT %Q* : FSOE_108803C1;
END_STRUCT
END_TYPE

// ---- DUTs/IO/PDOs/Module_1_FSOE_D19648F3.TcDUT
{attribute addProperty BoxType "EJ2914-0000-0017"}
{attribute addProperty Id "FSoE_InputsFSoE_Inputs_74C0DA41486FSoE_OutputsFSoE_Outputs_841EDA4B486"}
{attribute addProperty CRC "3516287219"}
{attribute addProperty SizeInBites "96"}
{attribute addProperty SizeInBytes "12"}
TYPE Module_1_FSOE_D19648F3 :
STRUCT
	{attribute addProperty Name "FSoE_Inputs"}
	FSoE_Inputs  : FSoE_Inputs_74C0DA41;
	{attribute addProperty Name "FSoE_Outputs"}
	FSoE_Outputs  : FSoE_Outputs_841EDA4B;
END_STRUCT
END_TYPE

// ---- DUTs/IO/PDOs/FSoE_Inputs_3EC5F4AF.TcDUT
{attribute addProperty BoxType "EJ2918-0000-0017"}
{attribute addProperty Id "FSOEAT %I*FSOE_E1AC8A65486"}
{attribute addProperty CRC "1053160623"}
{attribute addProperty SizeInBites "48"}
{attribute addProperty SizeInBytes "6"}
TYPE FSoE_Inputs_3EC5F4AF :
STRUCT
	{attribute addProperty Name "FSOE"}
	FSOE AT %I* : FSOE_E1AC8A65;
END_STRUCT
END_TYPE

// ---- DUTs/IO/PDOs/FSoE_Outputs_66F1C5B7.TcDUT
{attribute addProperty BoxType "EJ2918-0000-0017"}
{attribute addProperty Id "FSOEAT %Q*FSOE_89B9F66A567"}
{attribute addProperty CRC "1727120823"}
{attribute addProperty SizeInBites "56"}
{attribute addProperty SizeInBytes "7"}
TYPE FSoE_Outputs_66F1C5B7 :
STRUCT
	{attribute addProperty Name "FSOE"}
	FSOE AT %Q* : FSOE_89B9F66A;
END_STRUCT
END_TYPE

// ---- DUTs/IO/PDOs/Outputs_CA874E89.TcDUT
{attribute addProperty BoxType "EJ2918-0000-0017"}
{attribute addProperty Id "Module_1_Channel_1_Standard_OutputAT %Q*BOOL811Module_1_Channel_2_Standard_OutputAT %Q*BOOL812Module_1_Channel_3_Standard_OutputAT %Q*BOOL813Module_1_Channel_4_Standard_OutputAT %Q*BOOL814Module_2_Channel_1_Standard_OutputAT %Q*BOOL811Module_2_Channel_2_Standard_OutputAT %Q*BOOL812Module_2_Channel_3_Standard_OutputAT %Q*BOOL813Module_2_Channel_4_Standard_OutputAT %Q*BOOL814"}
{attribute addProperty CRC "3397865097"}
{attribute addProperty SizeInBites "64"}
{attribute addProperty SizeInBytes "8"}
TYPE Outputs_CA874E89 :
STRUCT
	{attribute addProperty Name "Module_1_Channel_1_Standard_Output"}
	Module_1_Channel_1_Standard_Output AT %Q* : BOOL;
	{attribute addProperty Name "Module_1_Channel_2_Standard_Output"}
	Module_1_Channel_2_Standard_Output AT %Q* : BOOL;
	{attribute addProperty Name "Module_1_Channel_3_Standard_Output"}
	Module_1_Channel_3_Standard_Output AT %Q* : BOOL;
	{attribute addProperty Name "Module_1_Channel_4_Standard_Output"}
	Module_1_Channel_4_Standard_Output AT %Q* : BOOL;
	{attribute addProperty Name "Module_2_Channel_1_Standard_Output"}
	Module_2_Channel_1_Standard_Output AT %Q* : BOOL;
	{attribute addProperty Name "Module_2_Channel_2_Standard_Output"}
	Module_2_Channel_2_Standard_Output AT %Q* : BOOL;
	{attribute addProperty Name "Module_2_Channel_3_Standard_Output"}
	Module_2_Channel_3_Standard_Output AT %Q* : BOOL;
	{attribute addProperty Name "Module_2_Channel_4_Standard_Output"}
	Module_2_Channel_4_Standard_Output AT %Q* : BOOL;
END_STRUCT
END_TYPE

// ---- DUTs/IO/PDOs/Module_1_FSOE_FC73D945.TcDUT
{attribute addProperty BoxType "EJ2918-0000-0017"}
{attribute addProperty Id "FSoE_InputsFSoE_Inputs_3EC5F4AF486FSoE_OutputsFSoE_Outputs_66F1C5B7567"}
{attribute addProperty CRC "4235450693"}
{attribute addProperty SizeInBites "104"}
{attribute addProperty SizeInBytes "13"}
TYPE Module_1_FSOE_FC73D945 :
STRUCT
	{attribute addProperty Name "FSoE_Inputs"}
	FSoE_Inputs  : FSoE_Inputs_3EC5F4AF;
	{attribute addProperty Name "FSoE_Outputs"}
	FSoE_Outputs  : FSoE_Outputs_66F1C5B7;
END_STRUCT
END_TYPE

// ---- DUTs/IO/PDOs/Module_2_FSOUT_15E08546.TcDUT
{attribute addProperty BoxType "EJ2918-0000-0017"}
{attribute addProperty Id "OutputsOutputs_CA874E89648"}
{attribute addProperty CRC "367035718"}
{attribute addProperty SizeInBites "64"}
{attribute addProperty SizeInBytes "8"}
TYPE Module_2_FSOUT_15E08546 :
STRUCT
	{attribute addProperty Name "Outputs"}
	Outputs  : Outputs_CA874E89;
END_STRUCT
END_TYPE

// ---- DUTs/IO/PDOs/InfoData_E9F65A82.TcDUT
{attribute addProperty BoxType "IODEVICETYPE_ETHERCATPROT"}
{attribute addProperty Id "ChangeCountAT %I*UINT1620DevIdAT %I*UINT1620AmsNetIdAT %I*AMSNETID4860CfgSlaveCountAT %I*UINT1620"}
{attribute addProperty CRC "3925236354"}
{attribute addProperty SizeInBites "96"}
{attribute addProperty SizeInBytes "12"}
TYPE InfoData_E9F65A82 :
STRUCT
	{attribute addProperty Name "ChangeCount"}
	ChangeCount AT %I* : UINT;
	{attribute addProperty Name "DevId"}
	DevId AT %I* : UINT;
	{attribute addProperty Name "AmsNetId"}
	AmsNetId AT %I* : AMSNETID;
	{attribute addProperty Name "CfgSlaveCount"}
	CfgSlaveCount AT %I* : UINT;
END_STRUCT
END_TYPE

// ---- DUTs/IO/PDOs/InfoData_BD06A15F.TcDUT
{attribute addProperty BoxType "IODEVICETYPE_ETHERCATPROT"}
{attribute addProperty Id "ObjectIdAT %I*OTCID3240StateAT %I*UINT1620SlaveCountAT %I*UINT1620"}
{attribute addProperty CRC "3171328351"}
{attribute addProperty SizeInBites "64"}
{attribute addProperty SizeInBytes "8"}
TYPE InfoData_BD06A15F :
STRUCT
	{attribute addProperty Name "ObjectId"}
	ObjectId AT %I* : OTCID;
	{attribute addProperty Name "State"}
	State AT %I* : UINT;
	{attribute addProperty Name "SlaveCount"}
	SlaveCount AT %I* : UINT;
END_STRUCT
END_TYPE

// ---- DUTs/IO/PDOs/Inputs_C3133F88.TcDUT
{attribute addProperty BoxType "IODEVICETYPE_ETHERCATPROT"}
{attribute addProperty Id "SlaveCountAT %I*UINT1620DevStateAT %I*UINT1620Frm0StateAT %I*UINT1620Frm0WcStateAT %I*UINT1620Frm0InputToggleAT %I*UINT1620Frm1StateAT %I*UINT1620Frm1WcStateAT %I*UINT1620Frm1InputToggleAT %I*UINT1620Frm2StateAT %I*UINT1620Frm2WcStateAT %I*UINT1620Frm2InputToggleAT %I*UINT1620Frm3StateAT %I*UINT1620Frm3WcStateAT %I*UINT1620Frm3InputToggleAT %I*UINT1620Frm4StateAT %I*UINT1620Frm4WcStateAT %I*UINT1620Frm4InputToggleAT %I*UINT1620Frm5StateAT %I*UINT1620Frm5WcStateAT %I*UINT1620Frm5InputToggleAT %I*UINT1620Frm6StateAT %I*UINT1620Frm6WcStateAT %I*UINT1620Frm6InputToggleAT %I*UINT1620Frm7StateAT %I*UINT1620Frm7WcStateAT %I*UINT1620Frm7InputToggleAT %I*UINT1620Frm8StateAT %I*UINT1620Frm8WcStateAT %I*UINT1620Frm8InputToggleAT %I*UINT1620Frm9StateAT %I*UINT1620Frm9WcStateAT %I*UINT1620Frm9InputToggleAT %I*UINT1620Frm10StateAT %I*UINT1620Frm10WcStateAT %I*UINT1620Frm10InputToggleAT %I*UINT1620Frm11StateAT %I*UINT1620Frm11WcStateAT %I*UINT1620Frm11InputToggleAT %I*UINT1620Frm12StateAT %I*UINT1620Frm12WcStateAT %I*UINT1620Frm12InputToggleAT %I*UINT1620Frm13StateAT %I*UINT1620Frm13WcStateAT %I*UINT1620Frm13InputToggleAT %I*UINT1620Frm14StateAT %I*UINT1620Frm14WcStateAT %I*UINT1620Frm14InputToggleAT %I*UINT1620Frm15StateAT %I*UINT1620Frm15WcStateAT %I*UINT1620Frm15InputToggleAT %I*UINT1620Frm16StateAT %I*UINT1620Frm16WcStateAT %I*UINT1620Frm16InputToggleAT %I*UINT1620Frm17StateAT %I*UINT1620Frm17WcStateAT %I*UINT1620Frm17InputToggleAT %I*UINT1620Frm18StateAT %I*UINT1620Frm18WcStateAT %I*UINT1620Frm18InputToggleAT %I*UINT1620Frm19StateAT %I*UINT1620Frm19WcStateAT %I*UINT1620Frm19InputToggleAT %I*UINT1620Frm20StateAT %I*UINT1620Frm20WcStateAT %I*UINT1620Frm20InputToggleAT %I*UINT1620Frm21StateAT %I*UINT1620Frm21WcStateAT %I*UINT1620Frm21InputToggleAT %I*UINT1620"}
{attribute addProperty CRC "3272818568"}
{attribute addProperty SizeInBites "1088"}
{attribute addProperty SizeInBytes "136"}
TYPE Inputs_C3133F88 :
STRUCT
	{attribute addProperty Name "SlaveCount"}
	SlaveCount AT %I* : UINT;
	{attribute addProperty Name "DevState"}
	DevState AT %I* : UINT;
	{attribute addProperty Name "Frm0State"}
	Frm0State AT %I* : UINT;
	{attribute addProperty Name "Frm0WcState"}
	Frm0WcState AT %I* : UINT;
	{attribute addProperty Name "Frm0InputToggle"}
	Frm0InputToggle AT %I* : UINT;
	{attribute addProperty Name "Frm1State"}
	Frm1State AT %I* : UINT;
	{attribute addProperty Name "Frm1WcState"}
	Frm1WcState AT %I* : UINT;
	{attribute addProperty Name "Frm1InputToggle"}
	Frm1InputToggle AT %I* : UINT;
	{attribute addProperty Name "Frm2State"}
	Frm2State AT %I* : UINT;
	{attribute addProperty Name "Frm2WcState"}
	Frm2WcState AT %I* : UINT;
	{attribute addProperty Name "Frm2InputToggle"}
	Frm2InputToggle AT %I* : UINT;
	{attribute addProperty Name "Frm3State"}
	Frm3State AT %I* : UINT;
	{attribute addProperty Name "Frm3WcState"}
	Frm3WcState AT %I* : UINT;
	{attribute addProperty Name "Frm3InputToggle"}
	Frm3InputToggle AT %I* : UINT;
	{attribute addProperty Name "Frm4State"}
	Frm4State AT %I* : UINT;
	{attribute addProperty Name "Frm4WcState"}
	Frm4WcState AT %I* : UINT;
	{attribute addProperty Name "Frm4InputToggle"}
	Frm4InputToggle AT %I* : UINT;
	{attribute addProperty Name "Frm5State"}
	Frm5State AT %I* : UINT;
	{attribute addProperty Name "Frm5WcState"}
	Frm5WcState AT %I* : UINT;
	{attribute addProperty Name "Frm5InputToggle"}
	Frm5InputToggle AT %I* : UINT;
	{attribute addProperty Name "Frm6State"}
	Frm6State AT %I* : UINT;
	{attribute addProperty Name "Frm6WcState"}
	Frm6WcState AT %I* : UINT;
	{attribute addProperty Name "Frm6InputToggle"}
	Frm6InputToggle AT %I* : UINT;
	{attribute addProperty Name "Frm7State"}
	Frm7State AT %I* : UINT;
	{attribute addProperty Name "Frm7WcState"}
	Frm7WcState AT %I* : UINT;
	{attribute addProperty Name "Frm7InputToggle"}
	Frm7InputToggle AT %I* : UINT;
	{attribute addProperty Name "Frm8State"}
	Frm8State AT %I* : UINT;
	{attribute addProperty Name "Frm8WcState"}
	Frm8WcState AT %I* : UINT;
	{attribute addProperty Name "Frm8InputToggle"}
	Frm8InputToggle AT %I* : UINT;
	{attribute addProperty Name "Frm9State"}
	Frm9State AT %I* : UINT;
	{attribute addProperty Name "Frm9WcState"}
	Frm9WcState AT %I* : UINT;
	{attribute addProperty Name "Frm9InputToggle"}
	Frm9InputToggle AT %I* : UINT;
	{attribute addProperty Name "Frm10State"}
	Frm10State AT %I* : UINT;
	{attribute addProperty Name "Frm10WcState"}
	Frm10WcState AT %I* : UINT;
	{attribute addProperty Name "Frm10InputToggle"}
	Frm10InputToggle AT %I* : UINT;
	{attribute addProperty Name "Frm11State"}
	Frm11State AT %I* : UINT;
	{attribute addProperty Name "Frm11WcState"}
	Frm11WcState AT %I* : UINT;
	{attribute addProperty Name "Frm11InputToggle"}
	Frm11InputToggle AT %I* : UINT;
	{attribute addProperty Name "Frm12State"}
	Frm12State AT %I* : UINT;
	{attribute addProperty Name "Frm12WcState"}
	Frm12WcState AT %I* : UINT;
	{attribute addProperty Name "Frm12InputToggle"}
	Frm12InputToggle AT %I* : UINT;
	{attribute addProperty Name "Frm13State"}
	Frm13State AT %I* : UINT;
	{attribute addProperty Name "Frm13WcState"}
	Frm13WcState AT %I* : UINT;
	{attribute addProperty Name "Frm13InputToggle"}
	Frm13InputToggle AT %I* : UINT;
	{attribute addProperty Name "Frm14State"}
	Frm14State AT %I* : UINT;
	{attribute addProperty Name "Frm14WcState"}
	Frm14WcState AT %I* : UINT;
	{attribute addProperty Name "Frm14InputToggle"}
	Frm14InputToggle AT %I* : UINT;
	{attribute addProperty Name "Frm15State"}
	Frm15State AT %I* : UINT;
	{attribute addProperty Name "Frm15WcState"}
	Frm15WcState AT %I* : UINT;
	{attribute addProperty Name "Frm15InputToggle"}
	Frm15InputToggle AT %I* : UINT;
	{attribute addProperty Name "Frm16State"}
	Frm16State AT %I* : UINT;
	{attribute addProperty Name "Frm16WcState"}
	Frm16WcState AT %I* : UINT;
	{attribute addProperty Name "Frm16InputToggle"}
	Frm16InputToggle AT %I* : UINT;
	{attribute addProperty Name "Frm17State"}
	Frm17State AT %I* : UINT;
	{attribute addProperty Name "Frm17WcState"}
	Frm17WcState AT %I* : UINT;
	{attribute addProperty Name "Frm17InputToggle"}
	Frm17InputToggle AT %I* : UINT;
	{attribute addProperty Name "Frm18State"}
	Frm18State AT %I* : UINT;
	{attribute addProperty Name "Frm18WcState"}
	Frm18WcState AT %I* : UINT;
	{attribute addProperty Name "Frm18InputToggle"}
	Frm18InputToggle AT %I* : UINT;
	{attribute addProperty Name "Frm19State"}
	Frm19State AT %I* : UINT;
	{attribute addProperty Name "Frm19WcState"}
	Frm19WcState AT %I* : UINT;
	{attribute addProperty Name "Frm19InputToggle"}
	Frm19InputToggle AT %I* : UINT;
	{attribute addProperty Name "Frm20State"}
	Frm20State AT %I* : UINT;
	{attribute addProperty Name "Frm20WcState"}
	Frm20WcState AT %I* : UINT;
	{attribute addProperty Name "Frm20InputToggle"}
	Frm20InputToggle AT %I* : UINT;
	{attribute addProperty Name "Frm21State"}
	Frm21State AT %I* : UINT;
	{attribute addProperty Name "Frm21WcState"}
	Frm21WcState AT %I* : UINT;
	{attribute addProperty Name "Frm21InputToggle"}
	Frm21InputToggle AT %I* : UINT;
END_STRUCT
END_TYPE

// ---- DUTs/IO/PDOs/Outputs_BAAAC746.TcDUT
{attribute addProperty BoxType "IODEVICETYPE_ETHERCATPROT"}
{attribute addProperty Id "DevCtrlAT %Q*UINT1620Frm0CtrlAT %Q*UINT1620Frm0WcCtrlAT %Q*UINT1620Frm1CtrlAT %Q*UINT1620Frm1WcCtrlAT %Q*UINT1620Frm2CtrlAT %Q*UINT1620Frm2WcCtrlAT %Q*UINT1620Frm3CtrlAT %Q*UINT1620Frm3WcCtrlAT %Q*UINT1620Frm4CtrlAT %Q*UINT1620Frm4WcCtrlAT %Q*UINT1620Frm5CtrlAT %Q*UINT1620Frm5WcCtrlAT %Q*UINT1620Frm6CtrlAT %Q*UINT1620Frm6WcCtrlAT %Q*UINT1620Frm7CtrlAT %Q*UINT1620Frm7WcCtrlAT %Q*UINT1620Frm8CtrlAT %Q*UINT1620Frm8WcCtrlAT %Q*UINT1620Frm9CtrlAT %Q*UINT1620Frm9WcCtrlAT %Q*UINT1620Frm10CtrlAT %Q*UINT1620Frm10WcCtrlAT %Q*UINT1620Frm11CtrlAT %Q*UINT1620Frm11WcCtrlAT %Q*UINT1620Frm12CtrlAT %Q*UINT1620Frm12WcCtrlAT %Q*UINT1620Frm13CtrlAT %Q*UINT1620Frm13WcCtrlAT %Q*UINT1620Frm14CtrlAT %Q*UINT1620Frm14WcCtrlAT %Q*UINT1620Frm15CtrlAT %Q*UINT1620Frm15WcCtrlAT %Q*UINT1620Frm16CtrlAT %Q*UINT1620Frm16WcCtrlAT %Q*UINT1620Frm17CtrlAT %Q*UINT1620Frm17WcCtrlAT %Q*UINT1620Frm18CtrlAT %Q*UINT1620Frm18WcCtrlAT %Q*UINT1620Frm19CtrlAT %Q*UINT1620Frm19WcCtrlAT %Q*UINT1620Frm20CtrlAT %Q*UINT1620Frm20WcCtrlAT %Q*UINT1620Frm21CtrlAT %Q*UINT1620Frm21WcCtrlAT %Q*UINT1620"}
{attribute addProperty CRC "3131754310"}
{attribute addProperty SizeInBites "720"}
{attribute addProperty SizeInBytes "90"}
TYPE Outputs_BAAAC746 :
STRUCT
	{attribute addProperty Name "DevCtrl"}
	DevCtrl AT %Q* : UINT;
	{attribute addProperty Name "Frm0Ctrl"}
	Frm0Ctrl AT %Q* : UINT;
	{attribute addProperty Name "Frm0WcCtrl"}
	Frm0WcCtrl AT %Q* : UINT;
	{attribute addProperty Name "Frm1Ctrl"}
	Frm1Ctrl AT %Q* : UINT;
	{attribute addProperty Name "Frm1WcCtrl"}
	Frm1WcCtrl AT %Q* : UINT;
	{attribute addProperty Name "Frm2Ctrl"}
	Frm2Ctrl AT %Q* : UINT;
	{attribute addProperty Name "Frm2WcCtrl"}
	Frm2WcCtrl AT %Q* : UINT;
	{attribute addProperty Name "Frm3Ctrl"}
	Frm3Ctrl AT %Q* : UINT;
	{attribute addProperty Name "Frm3WcCtrl"}
	Frm3WcCtrl AT %Q* : UINT;
	{attribute addProperty Name "Frm4Ctrl"}
	Frm4Ctrl AT %Q* : UINT;
	{attribute addProperty Name "Frm4WcCtrl"}
	Frm4WcCtrl AT %Q* : UINT;
	{attribute addProperty Name "Frm5Ctrl"}
	Frm5Ctrl AT %Q* : UINT;
	{attribute addProperty Name "Frm5WcCtrl"}
	Frm5WcCtrl AT %Q* : UINT;
	{attribute addProperty Name "Frm6Ctrl"}
	Frm6Ctrl AT %Q* : UINT;
	{attribute addProperty Name "Frm6WcCtrl"}
	Frm6WcCtrl AT %Q* : UINT;
	{attribute addProperty Name "Frm7Ctrl"}
	Frm7Ctrl AT %Q* : UINT;
	{attribute addProperty Name "Frm7WcCtrl"}
	Frm7WcCtrl AT %Q* : UINT;
	{attribute addProperty Name "Frm8Ctrl"}
	Frm8Ctrl AT %Q* : UINT;
	{attribute addProperty Name "Frm8WcCtrl"}
	Frm8WcCtrl AT %Q* : UINT;
	{attribute addProperty Name "Frm9Ctrl"}
	Frm9Ctrl AT %Q* : UINT;
	{attribute addProperty Name "Frm9WcCtrl"}
	Frm9WcCtrl AT %Q* : UINT;
	{attribute addProperty Name "Frm10Ctrl"}
	Frm10Ctrl AT %Q* : UINT;
	{attribute addProperty Name "Frm10WcCtrl"}
	Frm10WcCtrl AT %Q* : UINT;
	{attribute addProperty Name "Frm11Ctrl"}
	Frm11Ctrl AT %Q* : UINT;
	{attribute addProperty Name "Frm11WcCtrl"}
	Frm11WcCtrl AT %Q* : UINT;
	{attribute addProperty Name "Frm12Ctrl"}
	Frm12Ctrl AT %Q* : UINT;
	{attribute addProperty Name "Frm12WcCtrl"}
	Frm12WcCtrl AT %Q* : UINT;
	{attribute addProperty Name "Frm13Ctrl"}
	Frm13Ctrl AT %Q* : UINT;
	{attribute addProperty Name "Frm13WcCtrl"}
	Frm13WcCtrl AT %Q* : UINT;
	{attribute addProperty Name "Frm14Ctrl"}
	Frm14Ctrl AT %Q* : UINT;
	{attribute addProperty Name "Frm14WcCtrl"}
	Frm14WcCtrl AT %Q* : UINT;
	{attribute addProperty Name "Frm15Ctrl"}
	Frm15Ctrl AT %Q* : UINT;
	{attribute addProperty Name "Frm15WcCtrl"}
	Frm15WcCtrl AT %Q* : UINT;
	{attribute addProperty Name "Frm16Ctrl"}
	Frm16Ctrl AT %Q* : UINT;
	{attribute addProperty Name "Frm16WcCtrl"}
	Frm16WcCtrl AT %Q* : UINT;
	{attribute addProperty Name "Frm17Ctrl"}
	Frm17Ctrl AT %Q* : UINT;
	{attribute addProperty Name "Frm17WcCtrl"}
	Frm17WcCtrl AT %Q* : UINT;
	{attribute addProperty Name "Frm18Ctrl"}
	Frm18Ctrl AT %Q* : UINT;
	{attribute addProperty Name "Frm18WcCtrl"}
	Frm18WcCtrl AT %Q* : UINT;
	{attribute addProperty Name "Frm19Ctrl"}
	Frm19Ctrl AT %Q* : UINT;
	{attribute addProperty Name "Frm19WcCtrl"}
	Frm19WcCtrl AT %Q* : UINT;
	{attribute addProperty Name "Frm20Ctrl"}
	Frm20Ctrl AT %Q* : UINT;
	{attribute addProperty Name "Frm20WcCtrl"}
	Frm20WcCtrl AT %Q* : UINT;
	{attribute addProperty Name "Frm21Ctrl"}
	Frm21Ctrl AT %Q* : UINT;
	{attribute addProperty Name "Frm21WcCtrl"}
	Frm21WcCtrl AT %Q* : UINT;
END_STRUCT
END_TYPE

// ---- DUTs/IO/PDOs/ID_90FEAF08.TcDUT
{attribute addProperty BoxType "EK1101-0000-0016"}
{attribute addProperty Id "IDAT %I*UINT162"}
{attribute addProperty CRC "2432610056"}
{attribute addProperty SizeInBites "16"}
{attribute addProperty SizeInBytes "2"}
TYPE ID_90FEAF08 :
STRUCT
	{attribute addProperty Name "ID"}
	ID AT %I* : UINT;
END_STRUCT
END_TYPE

// ---- DUTs/IO/PDOs/Status_Us_D944C060.TcDUT
{attribute addProperty BoxType "EK1300-0000-0017"}
{attribute addProperty Id "UndervoltageAT %I*BOOL81"}
{attribute addProperty CRC "3645161568"}
{attribute addProperty SizeInBites "8"}
{attribute addProperty SizeInBytes "1"}
TYPE Status_Us_D944C060 :
STRUCT
	{attribute addProperty Name "Undervoltage"}
	Undervoltage AT %I* : BOOL;
END_STRUCT
END_TYPE

// ---- DUTs/IO/PDOs/Status_Up_D944C060.TcDUT
{attribute addProperty BoxType "EK1300-0000-0017"}
{attribute addProperty Id "UndervoltageAT %I*BOOL81"}
{attribute addProperty CRC "3645161568"}
{attribute addProperty SizeInBites "8"}
{attribute addProperty SizeInBytes "1"}
TYPE Status_Up_D944C060 :
STRUCT
	{attribute addProperty Name "Undervoltage"}
	Undervoltage AT %I* : BOOL;
END_STRUCT
END_TYPE

// ---- DUTs/IO/PDOs/MMS_Device_Inputs_EB48CD74.TcDUT
{attribute addProperty BoxType "EKM1101-0000-0016"}
{attribute addProperty Id "StatusAT %I*Status_BD85E94F162"}
{attribute addProperty CRC "3947416948"}
{attribute addProperty SizeInBites "16"}
{attribute addProperty SizeInBytes "2"}
TYPE MMS_Device_Inputs_EB48CD74 :
STRUCT
	{attribute addProperty Name "Status"}
	Status AT %I* : Status_BD85E94F;
END_STRUCT
END_TYPE

// ---- DUTs/IO/PDOs/MMS_Acceleration_Status_2FF1A472.TcDUT
{attribute addProperty BoxType "EKM1101-0000-0016"}
{attribute addProperty Id "StatusAT %I*Status_66D490D51621Number_of_samplesAT %I*UINT16217"}
{attribute addProperty CRC "804365426"}
{attribute addProperty SizeInBites "32"}
{attribute addProperty SizeInBytes "4"}
TYPE MMS_Acceleration_Status_2FF1A472 :
STRUCT
	{attribute addProperty Name "Status"}
	Status AT %I* : Status_66D490D5;
	{attribute addProperty Name "Number_of_samples"}
	Number_of_samples AT %I* : UINT;
END_STRUCT
END_TYPE

// ---- DUTs/IO/PDOs/MMS_Acceleration_X_Axis_2EF51F00.TcDUT
{attribute addProperty BoxType "EKM1101-0000-0016"}
{attribute addProperty Id "ValueAT %I*INT162"}
{attribute addProperty CRC "787816192"}
{attribute addProperty SizeInBites "16"}
{attribute addProperty SizeInBytes "2"}
TYPE MMS_Acceleration_X_Axis_2EF51F00 :
STRUCT
	{attribute addProperty Name "Value"}
	Value AT %I* : INT;
END_STRUCT
END_TYPE

// ---- DUTs/IO/PDOs/MMS_Acceleration_Y_Axis_2EF51F00.TcDUT
{attribute addProperty BoxType "EKM1101-0000-0016"}
{attribute addProperty Id "ValueAT %I*INT162"}
{attribute addProperty CRC "787816192"}
{attribute addProperty SizeInBites "16"}
{attribute addProperty SizeInBytes "2"}
TYPE MMS_Acceleration_Y_Axis_2EF51F00 :
STRUCT
	{attribute addProperty Name "Value"}
	Value AT %I* : INT;
END_STRUCT
END_TYPE

// ---- DUTs/IO/PDOs/MMS_Acceleration_Z_Axis_2EF51F00.TcDUT
{attribute addProperty BoxType "EKM1101-0000-0016"}
{attribute addProperty Id "ValueAT %I*INT162"}
{attribute addProperty CRC "787816192"}
{attribute addProperty SizeInBites "16"}
{attribute addProperty SizeInBytes "2"}
TYPE MMS_Acceleration_Z_Axis_2EF51F00 :
STRUCT
	{attribute addProperty Name "Value"}
	Value AT %I* : INT;
END_STRUCT
END_TYPE

// ---- DUTs/IO/PDOs/MMS_Acceleration_Timestamp_0B25C1A4.TcDUT
{attribute addProperty BoxType "EKM1101-0000-0016"}
{attribute addProperty Id "TimestampAT %I*ULINT648"}
{attribute addProperty CRC "187023780"}
{attribute addProperty SizeInBites "64"}
{attribute addProperty SizeInBytes "8"}
TYPE MMS_Acceleration_Timestamp_0B25C1A4 :
STRUCT
	{attribute addProperty Name "Timestamp"}
	Timestamp AT %I* : ULINT;
END_STRUCT
END_TYPE

// ---- DUTs/IO/PDOs/MMS_Voltage_Us_In_Inputs_BF33E0C1.TcDUT
{attribute addProperty BoxType "EKM1101-0000-0016"}
{attribute addProperty Id "StatusAT %I*Status_F0C7FE3C3241ValueAT %I*REAL32417"}
{attribute addProperty CRC "3207848129"}
{attribute addProperty SizeInBites "64"}
{attribute addProperty SizeInBytes "8"}
TYPE MMS_Voltage_Us_In_Inputs_BF33E0C1 :
STRUCT
	{attribute addProperty Name "Status"}
	Status AT %I* : Status_F0C7FE3C;
	{attribute addProperty Name "Value"}
	Value AT %I* : REAL;
END_STRUCT
END_TYPE

// ---- DUTs/IO/PDOs/MMS_Voltage_Up_In_Inputs_BF33E0C1.TcDUT
{attribute addProperty BoxType "EKM1101-0000-0016"}
{attribute addProperty Id "StatusAT %I*Status_F0C7FE3C3241ValueAT %I*REAL32417"}
{attribute addProperty CRC "3207848129"}
{attribute addProperty SizeInBites "64"}
{attribute addProperty SizeInBytes "8"}
TYPE MMS_Voltage_Up_In_Inputs_BF33E0C1 :
STRUCT
	{attribute addProperty Name "Status"}
	Status AT %I* : Status_F0C7FE3C;
	{attribute addProperty Name "Value"}
	Value AT %I* : REAL;
END_STRUCT
END_TYPE

// ---- DUTs/IO/PDOs/MMS_Voltage_Up_Out_Inputs_BF33E0C1.TcDUT
{attribute addProperty BoxType "EKM1101-0000-0016"}
{attribute addProperty Id "StatusAT %I*Status_F0C7FE3C3241ValueAT %I*REAL32417"}
{attribute addProperty CRC "3207848129"}
{attribute addProperty SizeInBites "64"}
{attribute addProperty SizeInBytes "8"}
TYPE MMS_Voltage_Up_Out_Inputs_BF33E0C1 :
STRUCT
	{attribute addProperty Name "Status"}
	Status AT %I* : Status_F0C7FE3C;
	{attribute addProperty Name "Value"}
	Value AT %I* : REAL;
END_STRUCT
END_TYPE

// ---- DUTs/IO/PDOs/MMS_Device_Outputs_39C15ABC.TcDUT
{attribute addProperty BoxType "EKM1101-0000-0016"}
{attribute addProperty Id "ControlAT %Q*Control_24A93024162"}
{attribute addProperty CRC "968972988"}
{attribute addProperty SizeInBites "16"}
{attribute addProperty SizeInBytes "2"}
TYPE MMS_Device_Outputs_39C15ABC :
STRUCT
	{attribute addProperty Name "Control"}
	Control AT %Q* : Control_24A93024;
END_STRUCT
END_TYPE

// ---- DUTs/IO/PDOs/InfoData_0BDED7BF.TcDUT
{attribute addProperty BoxType "EKM1101-0000-0016"}
{attribute addProperty Id "AdsAddrAT %I*AMSADDR6480DcOutputShiftAT %I*DINT3240DcInputShiftAT %I*DINT3240StateAT %I*UINT1620"}
{attribute addProperty CRC "199153599"}
{attribute addProperty SizeInBites "144"}
{attribute addProperty SizeInBytes "18"}
TYPE InfoData_0BDED7BF :
STRUCT
	{attribute addProperty Name "AdsAddr"}
	AdsAddr AT %I* : AMSADDR;
	{attribute addProperty Name "DcOutputShift"}
	DcOutputShift AT %I* : DINT;
	{attribute addProperty Name "DcInputShift"}
	DcInputShift AT %I* : DINT;
	{attribute addProperty Name "State"}
	State AT %I* : UINT;
END_STRUCT
END_TYPE

// ---- DUTs/IO/PDOs/FSoE_Inputs_FED5CD65.TcDUT
{attribute addProperty BoxType "EK1960-0000-0019"}
{attribute addProperty Id "FSOEAT %I*FSOE_F3ED5C6B12015"}
{attribute addProperty CRC "4275424613"}
{attribute addProperty SizeInBites "120"}
{attribute addProperty SizeInBytes "15"}
TYPE FSoE_Inputs_FED5CD65 :
STRUCT
	{attribute addProperty Name "FSOE"}
	FSOE AT %I* : FSOE_F3ED5C6B;
END_STRUCT
END_TYPE

// ---- DUTs/IO/PDOs/FSoE_Outputs_931DC9C5.TcDUT
{attribute addProperty BoxType "EK1960-0000-0019"}
{attribute addProperty Id "FSOEAT %Q*FSOE_B1AE0A9412015"}
{attribute addProperty CRC "2468202949"}
{attribute addProperty SizeInBites "120"}
{attribute addProperty SizeInBytes "15"}
TYPE FSoE_Outputs_931DC9C5 :
STRUCT
	{attribute addProperty Name "FSOE"}
	FSOE AT %Q* : FSOE_B1AE0A94;
END_STRUCT
END_TYPE

